LIN {X 0,Y 474.623,Z 516.173,A -85,B 0,C 180,E1 -7329.647,E2 -7329.647} C_VEL
LIN {X 0,Y 474.639,Z 516.177,A -85,B 0,C 180,E1 -7332.93,E2 -7332.93} C_VEL
LIN {X 0,Y 474.612,Z 516.174,A -85,B 0,C 180,E1 -7335.896,E2 -7335.896} C_VEL
LIN {X 0,Y 474.638,Z 516.178,A -85,B 0,C 180,E1 -7339.038,E2 -7339.038} C_VEL
LIN {X 0,Y 474.613,Z 516.174,A -85,B 0,C 180,E1 -7341.702,E2 -7341.702} C_VEL
LIN {X 0,Y 474.623,Z 516.175,A -85,B 0,C 180,E1 -7344.726,E2 -7344.726} C_VEL
LIN {X 0,Y 474.629,Z 516.17,A -85,B 0,C 180,E1 -7347.788,E2 -7347.788} C_VEL
LIN {X 0,Y 474.624,Z 516.176,A -85,B 0,C 180,E1 -7350.882,E2 -7350.882} C_VEL
LIN {X 0,Y 474.657,Z 516.166,A -85,B 0,C 180,E1 -7353.628,E2 -7353.628} C_VEL
LIN {X 0,Y 474.626,Z 516.176,A -85,B 0,C 180,E1 -7356.641,E2 -7356.641} C_VEL
LIN {X 0,Y 474.647,Z 516.168,A -85,B 0,C 180,E1 -7360.09,E2 -7360.09} C_VEL
LIN {X 0,Y 474.642,Z 516.174,A -85,B 0,C 180,E1 -7362.774,E2 -7362.774} C_VEL
LIN {X 0,Y 474.639,Z 516.173,A -85,B 0,C 180,E1 -7365.421,E2 -7365.421} C_VEL
LIN {X 0,Y 474.729,Z 516.161,A -85,B 0,C 180,E1 -7368.038,E2 -7368.038} C_VEL
LIN {X 0,Y 474.719,Z 516.164,A -85,B 0,C 180,E1 -7371.487,E2 -7371.487} C_VEL
LIN {X 0,Y 474.782,Z 516.155,A -85,B 0,C 180,E1 -7374.053,E2 -7374.053} C_VEL
LIN {X 0,Y 474.887,Z 516.143,A -85,B 0,C 180,E1 -7377.456,E2 -7377.456} C_VEL
LIN {X 0,Y 474.868,Z 516.149,A -85,B 0,C 180,E1 -7380.848,E2 -7380.848} C_VEL
LIN {X 0,Y 474.887,Z 516.145,A -85,B 0,C 180,E1 -7382.545,E2 -7382.545} C_VEL
LIN {X 0,Y 474.812,Z 516.337,A -85,B 0,C 180,E1 -7385.681,E2 -7385.681} C_VEL
LIN {X 0,Y 475.062,Z 517.484,A -85,B 0,C 180,E1 -7385.825,E2 -7385.825} C_VEL
LIN {X 0,Y 477.086,Z 523.784,A -85,B 0,C 180,E1 -7385.999,E2 -7385.999} C_VEL
LIN {X 0,Y 477.175,Z 549.292,A -85,B 0,C 180,E1 -7386.422,E2 -7386.422} C_VEL
LIN {X 0,Y 477.132,Z 562.414,A -85,B 0,C 180,E1 -7386.821,E2 -7386.821} C_VEL
LIN {X 0,Y 477,Z 574.255,A -85,B 0,C 180,E1 -7387.354,E2 -7387.354} C_VEL
LIN {X 0,Y 476.726,Z 585.813,A -85,B 0,C 180,E1 -7388.051,E2 -7388.051} C_VEL
LIN {X 0,Y 476.425,Z 597.212,A -85,B 0,C 180,E1 -7388.937,E2 -7388.937} C_VEL
LIN {X 0,Y 476.088,Z 605.867,A -85,B 0,C 180,E1 -7389.774,E2 -7389.774} C_VEL
LIN {X 0,Y 475.715,Z 614.993,A -85,B 0,C 180,E1 -7390.858,E2 -7390.858} C_VEL
LIN {X 0,Y 475.355,Z 623.876,A -85,B 0,C 180,E1 -7392.172,E2 -7392.172} C_VEL
LIN {X 0,Y 475.083,Z 630.832,A -85,B 0,C 180,E1 -7393.474,E2 -7393.474} C_VEL
LIN {X 0,Y 474.877,Z 635.577,A -85,B 0,C 180,E1 -7394.572,E2 -7394.572} C_VEL
LIN {X 0,Y 474.662,Z 639.7,A -85,B 0,C 180,E1 -7395.765,E2 -7395.765} C_VEL
LIN {X 0,Y 474.47,Z 643.459,A -85,B 0,C 180,E1 -7397.233,E2 -7397.233} C_VEL
LIN {X 0,Y 474.398,Z 645.704,A -85,B 0,C 180,E1 -7398.539,E2 -7398.539} C_VEL
LIN {X 0,Y 474.307,Z 647.024,A -85,B 0,C 180,E1 -7399.926,E2 -7399.926} C_VEL
LIN {X 0,Y 474.28,Z 647.331,A -85,B 0,C 180,E1 -7401.009,E2 -7401.009} C_VEL
LIN {X 0,Y 474.283,Z 647.161,A -85,B 0,C 180,E1 -7401.744,E2 -7401.744} C_VEL
LIN {X 0,Y 474.298,Z 645.84,A -85,B 0,C 180,E1 -7403.267,E2 -7403.267} C_VEL
LIN {X 0,Y 474.483,Z 642.883,A -85,B 0,C 180,E1 -7404.945,E2 -7404.945} C_VEL
LIN {X 0,Y 474.631,Z 639.027,A -85,B 0,C 180,E1 -7406.374,E2 -7406.374} C_VEL
LIN {X 0,Y 474.799,Z 633.826,A -85,B 0,C 180,E1 -7407.792,E2 -7407.792} C_VEL
LIN {X 0,Y 475.057,Z 627.036,A -85,B 0,C 180,E1 -7409.223,E2 -7409.223} C_VEL
LIN {X 0,Y 475.375,Z 619.877,A -85,B 0,C 180,E1 -7410.42,E2 -7410.42} C_VEL
LIN {X 0,Y 475.707,Z 610.882,A -85,B 0,C 180,E1 -7411.633,E2 -7411.633} C_VEL
LIN {X 0,Y 476.098,Z 600.971,A -85,B 0,C 180,E1 -7412.712,E2 -7412.712} C_VEL
LIN {X 0,Y 476.452,Z 591.039,A -85,B 0,C 180,E1 -7413.584,E2 -7413.584} C_VEL
LIN {X 0,Y 476.762,Z 579.896,A -85,B 0,C 180,E1 -7414.363,E2 -7414.363} C_VEL
LIN {X 0,Y 477.01,Z 567.71,A -85,B 0,C 180,E1 -7415.02,E2 -7415.02} C_VEL
LIN {X 0,Y 477.163,Z 555.29,A -85,B 0,C 180,E1 -7415.506,E2 -7415.506} C_VEL
LIN {X 0,Y 477.222,Z 541.716,A -85,B 0,C 180,E1 -7415.841,E2 -7415.841} C_VEL
LIN {X 0,Y 477.132,Z 524.228,A -85,B 0,C 180,E1 -7416.121,E2 -7416.121} C_VEL
LIN {X 0,Y 474.794,Z 517.041,A -85,B 0,C 180,E1 -7416.335,E2 -7416.335} C_VEL
LIN {X 0,Y 474.628,Z 516.233,A -85,B 0,C 180,E1 -7416.518,E2 -7416.518} C_VEL
LIN {X 0,Y 474.624,Z 516.178,A -85,B 0,C 180,E1 -7419.649,E2 -7419.649} C_VEL
LIN {X 0,Y 474.632,Z 516.175,A -85,B 0,C 180,E1 -7422.933,E2 -7422.933} C_VEL
LIN {X 0,Y 474.616,Z 516.174,A -85,B 0,C 180,E1 -7425.897,E2 -7425.897} C_VEL
LIN {X 0,Y 474.644,Z 516.172,A -85,B 0,C 180,E1 -7429.039,E2 -7429.039} C_VEL
LIN {X 0,Y 474.615,Z 516.177,A -85,B 0,C 180,E1 -7431.704,E2 -7431.704} C_VEL
LIN {X 0,Y 474.57,Z 516.182,A -85,B 0,C 180,E1 -7433.223,E2 -7433.223} C_VEL
LIN {X 0,Y 473.912,Z 516.264,A -85,B 0,C 180,E1 -7433.932,E2 -7433.932} C_VEL
LIN {X 0,Y 471.063,Z 516.618,A -85,B 0,C 180,E1 -7435.083,E2 -7435.083} C_VEL
LIN {X 0,Y 468.66,Z 516.916,A -85,B 0,C 180,E1 -7436.012,E2 -7436.012} C_VEL
LIN {X 0,Y 467.644,Z 517.042,A -85,B 0,C 180,E1 -7436.729,E2 -7436.729} C_VEL
LIN {X 0,Y 467.57,Z 517.052,A -85,B 0,C 180,E1 -7436.972,E2 -7436.972} C_VEL
LIN {X 0,Y 467.571,Z 517.055,A -85,B 0,C 180,E1 -7439.267,E2 -7439.267} C_VEL
LIN {X 0,Y 467.647,Z 517.04,A -85,B 0,C 180,E1 -7442.46,E2 -7442.46} C_VEL
LIN {X 0,Y 467.604,Z 517.049,A -85,B 0,C 180,E1 -7445.113,E2 -7445.113} C_VEL
LIN {X 0,Y 467.537,Z 517.057,A -85,B 0,C 180,E1 -7447.927,E2 -7447.927} C_VEL
LIN {X 0,Y 467.625,Z 517.043,A -85,B 0,C 180,E1 -7450.693,E2 -7450.693} C_VEL
LIN {X 0,Y 467.643,Z 517.042,A -85,B 0,C 180,E1 -7454.306,E2 -7454.306} C_VEL
LIN {X 0,Y 467.66,Z 517.044,A -85,B 0,C 180,E1 -7457.855,E2 -7457.855} C_VEL
LIN {X 0,Y 467.685,Z 517.04,A -85,B 0,C 180,E1 -7461.358,E2 -7461.358} C_VEL
LIN {X 0,Y 467.725,Z 517.035,A -85,B 0,C 180,E1 -7463.963,E2 -7463.963} C_VEL
LIN {X 0,Y 467.863,Z 517.018,A -85,B 0,C 180,E1 -7467.417,E2 -7467.417} C_VEL
LIN {X 0,Y 467.887,Z 517.015,A -85,B 0,C 180,E1 -7470,E2 -7470} C_VEL
LIN {X 0,Y 467.864,Z 517.013,A -85,B 0,C 180,E1 -7472.583,E2 -7472.583} C_VEL
LIN {X 0,Y 467.726,Z 517.036,A -85,B 0,C 180,E1 -7476.038,E2 -7476.038} C_VEL
LIN {X 0,Y 467.667,Z 517.042,A -85,B 0,C 180,E1 -7479.515,E2 -7479.515} C_VEL
LIN {X 0,Y 467.659,Z 517.041,A -85,B 0,C 180,E1 -7482.357,E2 -7482.357} C_VEL
LIN {X 0,Y 467.654,Z 517.048,A -85,B 0,C 180,E1 -7485.885,E2 -7485.885} C_VEL
LIN {X 0,Y 467.627,Z 517.044,A -85,B 0,C 180,E1 -7489.307,E2 -7489.307} C_VEL
LIN {X 0,Y 467.538,Z 517.06,A -85,B 0,C 180,E1 -7492.073,E2 -7492.073} C_VEL
LIN {X 0,Y 467.588,Z 517.048,A -85,B 0,C 180,E1 -7494.888,E2 -7494.888} C_VEL
LIN {X 0,Y 467.622,Z 517.049,A -85,B 0,C 180,E1 -7497.768,E2 -7497.768} C_VEL
LIN {X 0,Y 467.569,Z 517.05,A -85,B 0,C 180,E1 -7501.044,E2 -7501.044} C_VEL
LIN {X 0,Y 467.589,Z 517.053,A -85,B 0,C 180,E1 -7504.241,E2 -7504.241} C_VEL
LIN {X 0,Y 467.548,Z 517.053,A -85,B 0,C 180,E1 -7507.185,E2 -7507.185} C_VEL
LIN {X 0,Y 467.596,Z 517.053,A -85,B 0,C 180,E1 -7510.262,E2 -7510.262} C_VEL
LIN {X 0,Y 467.618,Z 517.046,A -85,B 0,C 180,E1 -7512.57,E2 -7512.57} C_VEL
LIN {X 0,Y 467.568,Z 517.05,A -85,B 0,C 180,E1 -7515.052,E2 -7515.052} C_VEL
LIN {X 0,Y 467.586,Z 517.049,A -85,B 0,C 180,E1 -7517.439,E2 -7517.439} C_VEL
LIN {X 0,Y 467.579,Z 517.05,A -85,B 0,C 180,E1 -7520.854,E2 -7520.854} C_VEL
LIN {X 0,Y 467.559,Z 517.059,A -85,B 0,C 180,E1 -7524.259,E2 -7524.259} C_VEL
LIN {X 0,Y 467.578,Z 517.049,A -85,B 0,C 180,E1 -7527.32,E2 -7527.32} C_VEL
LIN {X 0,Y 467.573,Z 517.052,A -85,B 0,C 180,E1 -7530.665,E2 -7530.665} C_VEL
LIN {X 0,Y 467.621,Z 517.043,A -85,B 0,C 180,E1 -7533.2,E2 -7533.2} C_VEL
LIN {X 0,Y 467.586,Z 517.054,A -85,B 0,C 180,E1 -7536.467,E2 -7536.467} C_VEL
LIN {X 0,Y 467.617,Z 517.046,A -85,B 0,C 180,E1 -7539.777,E2 -7539.777} C_VEL
LIN {X 0,Y 467.602,Z 517.052,A -85,B 0,C 180,E1 -7542.506,E2 -7542.506} C_VEL
LIN {X 0,Y 467.598,Z 517.047,A -85,B 0,C 180,E1 -7545.196,E2 -7545.196} C_VEL
LIN {X 0,Y 467.674,Z 517.039,A -85,B 0,C 180,E1 -7547.855,E2 -7547.855} C_VEL
LIN {X 0,Y 467.674,Z 517.037,A -85,B 0,C 180,E1 -7551.357,E2 -7551.357} C_VEL
LIN {X 0,Y 467.743,Z 517.031,A -85,B 0,C 180,E1 -7553.962,E2 -7553.962} C_VEL
LIN {X 0,Y 467.852,Z 517.015,A -85,B 0,C 180,E1 -7557.417,E2 -7557.417} C_VEL
LIN {X 0,Y 467.873,Z 517.014,A -85,B 0,C 180,E1 -7560,E2 -7560} C_VEL
LIN {X 0,Y 467.852,Z 517.022,A -85,B 0,C 180,E1 -7562.583,E2 -7562.583} C_VEL
LIN {X 0,Y 467.735,Z 517.032,A -85,B 0,C 180,E1 -7566.037,E2 -7566.037} C_VEL
LIN {X 0,Y 467.673,Z 517.044,A -85,B 0,C 180,E1 -7568.643,E2 -7568.643} C_VEL
LIN {X 0,Y 467.646,Z 517.043,A -85,B 0,C 180,E1 -7572.145,E2 -7572.145} C_VEL
LIN {X 0,Y 467.63,Z 517.042,A -85,B 0,C 180,E1 -7575.695,E2 -7575.695} C_VEL
LIN {X 0,Y 467.609,Z 517.052,A -85,B 0,C 180,E1 -7578.765,E2 -7578.765} C_VEL
LIN {X 0,Y 467.572,Z 517.051,A -85,B 0,C 180,E1 -7581.269,E2 -7581.269} C_VEL
LIN {X 0,Y 467.564,Z 517.051,A -85,B 0,C 180,E1 -7583.943,E2 -7583.943} C_VEL
LIN {X 0,Y 467.62,Z 517.051,A -85,B 0,C 180,E1 -7586.8,E2 -7586.8} C_VEL
LIN {X 0,Y 467.579,Z 517.049,A -85,B 0,C 180,E1 -7589.736,E2 -7589.736} C_VEL
LIN {X 0,Y 467.576,Z 517.058,A -85,B 0,C 180,E1 -7592.759,E2 -7592.759} C_VEL
LIN {X 0,Y 467.55,Z 517.052,A -85,B 0,C 180,E1 -7595.89,E2 -7595.89} C_VEL
LIN {X 0,Y 467.576,Z 517.053,A -85,B 0,C 180,E1 -7599.145,E2 -7599.145} C_VEL
LIN {X 0,Y 467.58,Z 517.053,A -85,B 0,C 180,E1 -7602.567,E2 -7602.567} C_VEL
LIN {X 0,Y 467.565,Z 517.056,A -85,B 0,C 180,E1 -7605.054,E2 -7605.054} C_VEL
LIN {X 0,Y 467.584,Z 517.05,A -85,B 0,C 180,E1 -7607.44,E2 -7607.44} C_VEL
LIN {X 0,Y 467.58,Z 517.057,A -85,B 0,C 180,E1 -7610.856,E2 -7610.856} C_VEL
LIN {X 0,Y 467.558,Z 517.054,A -85,B 0,C 180,E1 -7614.261,E2 -7614.261} C_VEL
LIN {X 0,Y 467.579,Z 517.057,A -85,B 0,C 180,E1 -7617.321,E2 -7617.321} C_VEL
LIN {X 0,Y 467.62,Z 517.228,A -85,B 0,C 180,E1 -7618.944,E2 -7618.944} C_VEL
LIN {X 0,Y 470.423,Z 531.107,A -85,B 0,C 180,E1 -7621.678,E2 -7621.678} C_VEL
LIN {X 0,Y 470.116,Z 540.418,A -85,B 0,C 180,E1 -7623.354,E2 -7623.354} C_VEL
LIN {X 0,Y 469.299,Z 558.979,A -85,B 0,C 180,E1 -7626.619,E2 -7626.619} C_VEL
LIN {X 0,Y 468.488,Z 577.522,A -85,B 0,C 180,E1 -7629.817,E2 -7629.817} C_VEL
LIN {X 0,Y 468.046,Z 592.113,A -85,B 0,C 180,E1 -7632.298,E2 -7632.298} C_VEL
LIN {X 0,Y 467.637,Z 610.659,A -85,B 0,C 180,E1 -7635.42,E2 -7635.42} C_VEL
LIN {X 0,Y 467.447,Z 616.633,A -85,B 0,C 180,E1 -7636.386,E2 -7636.386} C_VEL
LIN {X 0,Y 469.563,Z 640.275,A -85,B 0,C 180,E1 -7636.878,E2 -7636.878} C_VEL
LIN {X 0,Y 469.124,Z 698.067,A -85,B 0,C 180,E1 -7637.871,E2 -7637.871} C_VEL
LIN {X 0,Y 468.748,Z 709.114,A -85,B 0,C 180,E1 -7638.213,E2 -7638.213} C_VEL
LIN {X 0,Y 468.397,Z 720.606,A -85,B 0,C 180,E1 -7638.752,E2 -7638.752} C_VEL
LIN {X 0,Y 468.018,Z 730.817,A -85,B 0,C 180,E1 -7639.4,E2 -7639.4} C_VEL
LIN {X 0,Y 467.616,Z 741.243,A -85,B 0,C 180,E1 -7640.266,E2 -7640.266} C_VEL
LIN {X 0,Y 467.318,Z 749.497,A -85,B 0,C 180,E1 -7641.133,E2 -7641.133} C_VEL
LIN {X 0,Y 467.121,Z 757.771,A -85,B 0,C 180,E1 -7642.218,E2 -7642.218} C_VEL
LIN {X 0,Y 467.063,Z 764.185,A -85,B 0,C 180,E1 -7643.272,E2 -7643.272} C_VEL
LIN {X 0,Y 466.964,Z 769.568,A -85,B 0,C 180,E1 -7644.386,E2 -7644.386} C_VEL
LIN {X 0,Y 466.953,Z 774.391,A -85,B 0,C 180,E1 -7645.684,E2 -7645.684} C_VEL
LIN {X 0,Y 466.975,Z 776.783,A -85,B 0,C 180,E1 -7646.549,E2 -7646.549} C_VEL
LIN {X 0,Y 466.93,Z 778.604,A -85,B 0,C 180,E1 -7647.412,E2 -7647.412} C_VEL
LIN {X 0,Y 466.913,Z 779.879,A -85,B 0,C 180,E1 -7648.275,E2 -7648.275} C_VEL
LIN {X 0,Y 466.917,Z 780.608,A -85,B 0,C 180,E1 -7649.138,E2 -7649.138} C_VEL
LIN {X 0,Y 467.053,Z 780.859,A -85,B 0,C 180,E1 -7650,E2 -7650} C_VEL
LIN {X 0,Y 466.929,Z 780.514,A -85,B 0,C 180,E1 -7650.862,E2 -7650.862} C_VEL
LIN {X 0,Y 466.936,Z 779.7,A -85,B 0,C 180,E1 -7651.725,E2 -7651.725} C_VEL
LIN {X 0,Y 466.961,Z 778.321,A -85,B 0,C 180,E1 -7652.588,E2 -7652.588} C_VEL
LIN {X 0,Y 467.012,Z 775.24,A -85,B 0,C 180,E1 -7653.883,E2 -7653.883} C_VEL
LIN {X 0,Y 466.958,Z 770.741,A -85,B 0,C 180,E1 -7655.181,E2 -7655.181} C_VEL
LIN {X 0,Y 467.062,Z 764.905,A -85,B 0,C 180,E1 -7656.445,E2 -7656.445} C_VEL
LIN {X 0,Y 467.113,Z 758.249,A -85,B 0,C 180,E1 -7657.565,E2 -7657.565} C_VEL
LIN {X 0,Y 467.283,Z 750.162,A -85,B 0,C 180,E1 -7658.65,E2 -7658.65} C_VEL
LIN {X 0,Y 467.545,Z 740.997,A -85,B 0,C 180,E1 -7659.626,E2 -7659.626} C_VEL
LIN {X 0,Y 467.91,Z 730.624,A -85,B 0,C 180,E1 -7660.493,E2 -7660.493} C_VEL
LIN {X 0,Y 468.299,Z 719.691,A -85,B 0,C 180,E1 -7661.195,E2 -7661.195} C_VEL
LIN {X 0,Y 468.652,Z 708.238,A -85,B 0,C 180,E1 -7661.735,E2 -7661.735} C_VEL
LIN {X 0,Y 469.06,Z 696.256,A -85,B 0,C 180,E1 -7662.108,E2 -7662.108} C_VEL
LIN {X 0,Y 469.386,Z 644.85,A -85,B 0,C 180,E1 -7662.978,E2 -7662.978} C_VEL
LIN {X 0,Y 469.097,Z 635.875,A -85,B 0,C 180,E1 -7663.138,E2 -7663.138} C_VEL
LIN {X 0,Y 467.424,Z 613.413,A -85,B 0,C 180,E1 -7663.587,E2 -7663.587} C_VEL
LIN {X 0,Y 467.456,Z 610.902,A -85,B 0,C 180,E1 -7663.919,E2 -7663.919} C_VEL
LIN {X 0,Y 467.813,Z 590.403,A -85,B 0,C 180,E1 -7667.259,E2 -7667.259} C_VEL
LIN {X 0,Y 468.259,Z 569.924,A -85,B 0,C 180,E1 -7670.652,E2 -7670.652} C_VEL
LIN {X 0,Y 468.806,Z 550.911,A -85,B 0,C 180,E1 -7673.876,E2 -7673.876} C_VEL
LIN {X 0,Y 469.473,Z 532.108,A -85,B 0,C 180,E1 -7677.166,E2 -7677.166} C_VEL
LIN {X 0,Y 469.564,Z 527.557,A -85,B 0,C 180,E1 -7677.987,E2 -7677.987} C_VEL
LIN {X 0,Y 467.63,Z 517.169,A -85,B 0,C 180,E1 -7680.042,E2 -7680.042} C_VEL
LIN {X 0,Y 467.58,Z 517.056,A -85,B 0,C 180,E1 -7682.758,E2 -7682.758} C_VEL
LIN {X 0,Y 467.551,Z 517.055,A -85,B 0,C 180,E1 -7685.889,E2 -7685.889} C_VEL
LIN {X 0,Y 467.578,Z 517.056,A -85,B 0,C 180,E1 -7689.144,E2 -7689.144} C_VEL
LIN {X 0,Y 467.58,Z 517.052,A -85,B 0,C 180,E1 -7692.566,E2 -7692.566} C_VEL
LIN {X 0,Y 467.564,Z 517.056,A -85,B 0,C 180,E1 -7695.053,E2 -7695.053} C_VEL
LIN {X 0,Y 467.618,Z 517.044,A -85,B 0,C 180,E1 -7697.443,E2 -7697.443} C_VEL
LIN {X 0,Y 467.612,Z 517.049,A -85,B 0,C 180,E1 -7700.858,E2 -7700.858} C_VEL
LIN {X 0,Y 467.556,Z 517.052,A -85,B 0,C 180,E1 -7704.26,E2 -7704.26} C_VEL
LIN {X 0,Y 467.574,Z 517.052,A -85,B 0,C 180,E1 -7707.32,E2 -7707.32} C_VEL
LIN {X 0,Y 467.57,Z 517.054,A -85,B 0,C 180,E1 -7710.665,E2 -7710.665} C_VEL
LIN {X 0,Y 467.619,Z 517.046,A -85,B 0,C 180,E1 -7713.2,E2 -7713.2} C_VEL
LIN {X 0,Y 467.583,Z 517.052,A -85,B 0,C 180,E1 -7716.468,E2 -7716.468} C_VEL
LIN {X 0,Y 467.614,Z 517.044,A -85,B 0,C 180,E1 -7719.777,E2 -7719.777} C_VEL
LIN {X 0,Y 467.6,Z 517.05,A -85,B 0,C 180,E1 -7722.507,E2 -7722.507} C_VEL
LIN {X 0,Y 467.597,Z 517.053,A -85,B 0,C 180,E1 -7725.196,E2 -7725.196} C_VEL
LIN {X 0,Y 467.687,Z 517.038,A -85,B 0,C 180,E1 -7727.856,E2 -7727.856} C_VEL
LIN {X 0,Y 467.673,Z 517.043,A -85,B 0,C 180,E1 -7731.357,E2 -7731.357} C_VEL
LIN {X 0,Y 467.744,Z 517.032,A -85,B 0,C 180,E1 -7733.963,E2 -7733.963} C_VEL
LIN {X 0,Y 467.852,Z 517.02,A -85,B 0,C 180,E1 -7737.417,E2 -7737.417} C_VEL
LIN {X 0,Y 467.873,Z 517.016,A -85,B 0,C 180,E1 -7740,E2 -7740} C_VEL
LIN {X 0,Y 467.852,Z 517.021,A -85,B 0,C 180,E1 -7742.583,E2 -7742.583} C_VEL
LIN {X 0,Y 467.76,Z 517.165,A -85,B 0,C 180,E1 -7745.443,E2 -7745.443} C_VEL
LIN {X 0,Y 467.998,Z 518.237,A -85,B 0,C 180,E1 -7745.602,E2 -7745.602} C_VEL
LIN {X 0,Y 470.331,Z 525.484,A -85,B 0,C 180,E1 -7745.803,E2 -7745.803} C_VEL
LIN {X 0,Y 470.316,Z 550.256,A -85,B 0,C 180,E1 -7746.22,E2 -7746.22} C_VEL
LIN {X 0,Y 470.277,Z 563.453,A -85,B 0,C 180,E1 -7746.624,E2 -7746.624} C_VEL
LIN {X 0,Y 470.145,Z 575.827,A -85,B 0,C 180,E1 -7747.192,E2 -7747.192} C_VEL
LIN {X 0,Y 469.824,Z 588.1,A -85,B 0,C 180,E1 -7747.954,E2 -7747.954} C_VEL
LIN {X 0,Y 469.566,Z 598.1,A -85,B 0,C 180,E1 -7748.752,E2 -7748.752} C_VEL
LIN {X 0,Y 469.156,Z 607.733,A -85,B 0,C 180,E1 -7749.702,E2 -7749.702} C_VEL
LIN {X 0,Y 468.807,Z 616.704,A -85,B 0,C 180,E1 -7750.801,E2 -7750.801} C_VEL
LIN {X 0,Y 468.4,Z 625.436,A -85,B 0,C 180,E1 -7752.126,E2 -7752.126} C_VEL
LIN {X 0,Y 468.104,Z 632.319,A -85,B 0,C 180,E1 -7753.457,E2 -7753.457} C_VEL
LIN {X 0,Y 467.852,Z 637.784,A -85,B 0,C 180,E1 -7754.796,E2 -7754.796} C_VEL
LIN {X 0,Y 467.635,Z 641.308,A -85,B 0,C 180,E1 -7755.883,E2 -7755.883} C_VEL
LIN {X 0,Y 467.454,Z 645.129,A -85,B 0,C 180,E1 -7757.5,E2 -7757.5} C_VEL
LIN {X 0,Y 467.376,Z 646.948,A -85,B 0,C 180,E1 -7758.681,E2 -7758.681} C_VEL
LIN {X 0,Y 467.289,Z 648.199,A -85,B 0,C 180,E1 -7760.238,E2 -7760.238} C_VEL
LIN {X 0,Y 467.263,Z 648.317,A -85,B 0,C 180,E1 -7761.171,E2 -7761.171} C_VEL
LIN {X 0,Y 467.254,Z 647.963,A -85,B 0,C 180,E1 -7762.088,E2 -7762.088} C_VEL
LIN {X 0,Y 467.285,Z 646.625,A -85,B 0,C 180,E1 -7763.448,E2 -7763.448} C_VEL
LIN {X 0,Y 467.451,Z 644.073,A -85,B 0,C 180,E1 -7764.896,E2 -7764.896} C_VEL
LIN {X 0,Y 467.619,Z 640.383,A -85,B 0,C 180,E1 -7766.319,E2 -7766.319} C_VEL
LIN {X 0,Y 467.806,Z 635.294,A -85,B 0,C 180,E1 -7767.757,E2 -7767.757} C_VEL
LIN {X 0,Y 468.037,Z 629.218,A -85,B 0,C 180,E1 -7769.09,E2 -7769.09} C_VEL
LIN {X 0,Y 468.386,Z 621.573,A -85,B 0,C 180,E1 -7770.425,E2 -7770.425} C_VEL
LIN {X 0,Y 468.74,Z 612.773,A -85,B 0,C 180,E1 -7771.653,E2 -7771.653} C_VEL
LIN {X 0,Y 469.139,Z 602.841,A -85,B 0,C 180,E1 -7772.767,E2 -7772.767} C_VEL
LIN {X 0,Y 469.496,Z 593.334,A -85,B 0,C 180,E1 -7773.633,E2 -7773.633} C_VEL
LIN {X 0,Y 469.831,Z 581.764,A -85,B 0,C 180,E1 -7774.475,E2 -7774.475} C_VEL
LIN {X 0,Y 470.109,Z 569.848,A -85,B 0,C 180,E1 -7775.139,E2 -7775.139} C_VEL
LIN {X 0,Y 470.277,Z 556.846,A -85,B 0,C 180,E1 -7775.669,E2 -7775.669} C_VEL
LIN {X 0,Y 470.314,Z 543.458,A -85,B 0,C 180,E1 -7776.013,E2 -7776.013} C_VEL
LIN {X 0,Y 470.23,Z 525.469,A -85,B 0,C 180,E1 -7776.312,E2 -7776.312} C_VEL
LIN {X 0,Y 467.743,Z 517.998,A -85,B 0,C 180,E1 -7776.528,E2 -7776.528} C_VEL
LIN {X 0,Y 467.563,Z 517.133,A -85,B 0,C 180,E1 -7776.701,E2 -7776.701} C_VEL
LIN {X 0,Y 467.579,Z 517.054,A -85,B 0,C 180,E1 -7779.956,E2 -7779.956} C_VEL
LIN {X 0,Y 467.583,Z 517.051,A -85,B 0,C 180,E1 -7782.568,E2 -7782.568} C_VEL
LIN {X 0,Y 467.568,Z 517.054,A -85,B 0,C 180,E1 -7785.054,E2 -7785.054} C_VEL
LIN {X 0,Y 467.622,Z 517.051,A -85,B 0,C 180,E1 -7787.445,E2 -7787.445} C_VEL
LIN {X 0,Y 467.614,Z 517.046,A -85,B 0,C 180,E1 -7790.86,E2 -7790.86} C_VEL
LIN {X 0,Y 467.559,Z 517.052,A -85,B 0,C 180,E1 -7794.262,E2 -7794.262} C_VEL
LIN {X 0,Y 467.57,Z 517.052,A -85,B 0,C 180,E1 -7796.972,E2 -7796.972} C_VEL
LIN {X 0,Y 466.932,Z 517.138,A -85,B 0,C 180,E1 -7797.69,E2 -7797.69} C_VEL
LIN {X 0,Y 464.104,Z 517.49,A -85,B 0,C 180,E1 -7798.857,E2 -7798.857} C_VEL
LIN {X 0,Y 461.688,Z 517.788,A -85,B 0,C 180,E1 -7799.798,E2 -7799.798} C_VEL
LIN {X 0,Y 460.634,Z 517.916,A -85,B 0,C 180,E1 -7800.525,E2 -7800.525} C_VEL
LIN {X 0,Y 460.541,Z 517.926,A -85,B 0,C 180,E1 -7800.771,E2 -7800.771} C_VEL
LIN {X 0,Y 460.565,Z 517.928,A -85,B 0,C 180,E1 -7803.736,E2 -7803.736} C_VEL
LIN {X 0,Y 460.548,Z 517.925,A -85,B 0,C 180,E1 -7806.625,E2 -7806.625} C_VEL
LIN {X 0,Y 460.554,Z 517.931,A -85,B 0,C 180,E1 -7809.453,E2 -7809.453} C_VEL
LIN {X 0,Y 460.553,Z 517.925,A -85,B 0,C 180,E1 -7812.23,E2 -7812.23} C_VEL
LIN {X 0,Y 460.569,Z 517.923,A -85,B 0,C 180,E1 -7814.965,E2 -7814.965} C_VEL
LIN {X 0,Y 460.615,Z 517.916,A -85,B 0,C 180,E1 -7818.56,E2 -7818.56} C_VEL
LIN {X 0,Y 460.671,Z 517.912,A -85,B 0,C 180,E1 -7822.108,E2 -7822.108} C_VEL
LIN {X 0,Y 460.693,Z 517.906,A -85,B 0,C 180,E1 -7824.748,E2 -7824.748} C_VEL
LIN {X 0,Y 460.804,Z 517.897,A -85,B 0,C 180,E1 -7827.378,E2 -7827.378} C_VEL
LIN {X 0,Y 460.858,Z 517.891,A -85,B 0,C 180,E1 -7830,E2 -7830} C_VEL
LIN {X 0,Y 460.805,Z 517.893,A -85,B 0,C 180,E1 -7832.622,E2 -7832.622} C_VEL
LIN {X 0,Y 460.69,Z 517.911,A -85,B 0,C 180,E1 -7836.13,E2 -7836.13} C_VEL
LIN {X 0,Y 460.625,Z 517.915,A -85,B 0,C 180,E1 -7838.776,E2 -7838.776} C_VEL
LIN {X 0,Y 460.618,Z 517.917,A -85,B 0,C 180,E1 -7842.445,E2 -7842.445} C_VEL
LIN {X 0,Y 460.604,Z 517.924,A -85,B 0,C 180,E1 -7845.997,E2 -7845.997} C_VEL
LIN {X 0,Y 460.575,Z 517.921,A -85,B 0,C 180,E1 -7848.901,E2 -7848.901} C_VEL
LIN {X 0,Y 460.519,Z 517.931,A -85,B 0,C 180,E1 -7851.485,E2 -7851.485} C_VEL
LIN {X 0,Y 460.534,Z 517.93,A -85,B 0,C 180,E1 -7854.332,E2 -7854.332} C_VEL
LIN {X 0,Y 460.573,Z 517.922,A -85,B 0,C 180,E1 -7857.243,E2 -7857.243} C_VEL
LIN {X 0,Y 460.512,Z 517.934,A -85,B 0,C 180,E1 -7860.239,E2 -7860.239} C_VEL
LIN {X 0,Y 460.53,Z 517.928,A -85,B 0,C 180,E1 -7863.324,E2 -7863.324} C_VEL
LIN {X 0,Y 460.476,Z 517.936,A -85,B 0,C 180,E1 -7866.529,E2 -7866.529} C_VEL
LIN {X 0,Y 460.574,Z 517.927,A -85,B 0,C 180,E1 -7869.857,E2 -7869.857} C_VEL
LIN {X 0,Y 460.541,Z 517.926,A -85,B 0,C 180,E1 -7872.903,E2 -7872.903} C_VEL
LIN {X 0,Y 460.509,Z 517.934,A -85,B 0,C 180,E1 -7875.829,E2 -7875.829} C_VEL
LIN {X 0,Y 460.528,Z 517.927,A -85,B 0,C 180,E1 -7878.988,E2 -7878.988} C_VEL
LIN {X 0,Y 460.523,Z 517.928,A -85,B 0,C 180,E1 -7881.266,E2 -7881.266} C_VEL
LIN {X 0,Y 460.509,Z 517.933,A -85,B 0,C 180,E1 -7884.554,E2 -7884.554} C_VEL
LIN {X 0,Y 460.528,Z 517.929,A -85,B 0,C 180,E1 -7887.715,E2 -7887.715} C_VEL
LIN {X 0,Y 460.542,Z 517.927,A -85,B 0,C 180,E1 -7890.769,E2 -7890.769} C_VEL
LIN {X 0,Y 460.562,Z 517.925,A -85,B 0,C 180,E1 -7893.734,E2 -7893.734} C_VEL
LIN {X 0,Y 460.539,Z 517.93,A -85,B 0,C 180,E1 -7896.623,E2 -7896.623} C_VEL
LIN {X 0,Y 460.545,Z 517.925,A -85,B 0,C 180,E1 -7899.452,E2 -7899.452} C_VEL
LIN {X 0,Y 460.552,Z 517.931,A -85,B 0,C 180,E1 -7902.23,E2 -7902.23} C_VEL
LIN {X 0,Y 460.557,Z 517.925,A -85,B 0,C 180,E1 -7904.964,E2 -7904.964} C_VEL
LIN {X 0,Y 460.621,Z 517.916,A -85,B 0,C 180,E1 -7907.666,E2 -7907.666} C_VEL
LIN {X 0,Y 460.621,Z 517.916,A -85,B 0,C 180,E1 -7911.223,E2 -7911.223} C_VEL
LIN {X 0,Y 460.708,Z 517.906,A -85,B 0,C 180,E1 -7913.87,E2 -7913.87} C_VEL
LIN {X 0,Y 460.817,Z 517.891,A -85,B 0,C 180,E1 -7917.377,E2 -7917.377} C_VEL
LIN {X 0,Y 460.844,Z 517.89,A -85,B 0,C 180,E1 -7920,E2 -7920} C_VEL
LIN {X 0,Y 460.817,Z 517.898,A -85,B 0,C 180,E1 -7922.622,E2 -7922.622} C_VEL
LIN {X 0,Y 460.701,Z 517.909,A -85,B 0,C 180,E1 -7926.13,E2 -7926.13} C_VEL
LIN {X 0,Y 460.62,Z 517.921,A -85,B 0,C 180,E1 -7928.776,E2 -7928.776} C_VEL
LIN {X 0,Y 460.604,Z 517.924,A -85,B 0,C 180,E1 -7932.445,E2 -7932.445} C_VEL
LIN {X 0,Y 460.591,Z 517.92,A -85,B 0,C 180,E1 -7935.998,E2 -7935.998} C_VEL
LIN {X 0,Y 460.562,Z 517.928,A -85,B 0,C 180,E1 -7938.902,E2 -7938.902} C_VEL
LIN {X 0,Y 460.507,Z 517.93,A -85,B 0,C 180,E1 -7941.486,E2 -7941.486} C_VEL
LIN {X 0,Y 460.534,Z 517.93,A -85,B 0,C 180,E1 -7944.332,E2 -7944.332} C_VEL
LIN {X 0,Y 460.576,Z 517.923,A -85,B 0,C 180,E1 -7947.243,E2 -7947.243} C_VEL
LIN {X 0,Y 460.52,Z 517.93,A -85,B 0,C 180,E1 -7950.239,E2 -7950.239} C_VEL
LIN {X 0,Y 460.522,Z 517.93,A -85,B 0,C 180,E1 -7953.325,E2 -7953.325} C_VEL
LIN {X 0,Y 460.472,Z 517.939,A -85,B 0,C 180,E1 -7956.53,E2 -7956.53} C_VEL
LIN {X 0,Y 460.538,Z 517.933,A -85,B 0,C 180,E1 -7958.898,E2 -7958.898} C_VEL
LIN {X 0,Y 460.518,Z 517.929,A -85,B 0,C 180,E1 -7962.182,E2 -7962.182} C_VEL
LIN {X 0,Y 460.515,Z 517.93,A -85,B 0,C 180,E1 -7965.412,E2 -7965.412} C_VEL
LIN {X 0,Y 460.53,Z 517.929,A -85,B 0,C 180,E1 -7968.398,E2 -7968.398} C_VEL
LIN {X 0,Y 460.527,Z 517.931,A -85,B 0,C 180,E1 -7971.268,E2 -7971.268} C_VEL
LIN {X 0,Y 460.509,Z 517.935,A -85,B 0,C 180,E1 -7974.555,E2 -7974.555} C_VEL
LIN {X 0,Y 460.532,Z 517.933,A -85,B 0,C 180,E1 -7977.716,E2 -7977.716} C_VEL
LIN {X 0,Y 460.579,Z 518.159,A -85,B 0,C 180,E1 -7978.748,E2 -7978.748} C_VEL
LIN {X 0,Y 463.448,Z 532.352,A -85,B 0,C 180,E1 -7981.587,E2 -7981.587} C_VEL
LIN {X 0,Y 463.28,Z 539.644,A -85,B 0,C 180,E1 -7982.929,E2 -7982.929} C_VEL
LIN {X 0,Y 462.298,Z 559.467,A -85,B 0,C 180,E1 -7986.481,E2 -7986.481} C_VEL
LIN {X 0,Y 461.458,Z 577.955,A -85,B 0,C 180,E1 -7989.728,E2 -7989.728} C_VEL
LIN {X 0,Y 460.904,Z 595.124,A -85,B 0,C 180,E1 -7992.702,E2 -7992.702} C_VEL
LIN {X 0,Y 460.409,Z 613.57,A -85,B 0,C 180,E1 -7995.864,E2 -7995.864} C_VEL
LIN {X 0,Y 460.41,Z 615.765,A -85,B 0,C 180,E1 -7996.173,E2 -7996.173} C_VEL
LIN {X 0,Y 462.655,Z 641.477,A -85,B 0,C 180,E1 -7996.704,E2 -7996.704} C_VEL
LIN {X 0,Y 462.148,Z 697.14,A -85,B 0,C 180,E1 -7997.685,E2 -7997.685} C_VEL
LIN {X 0,Y 461.79,Z 708.124,A -85,B 0,C 180,E1 -7998.033,E2 -7998.033} C_VEL
LIN {X 0,Y 461.414,Z 719.591,A -85,B 0,C 180,E1 -7998.58,E2 -7998.58} C_VEL
LIN {X 0,Y 461.027,Z 729.799,A -85,B 0,C 180,E1 -7999.238,E2 -7999.238} C_VEL
LIN {X 0,Y 460.621,Z 740.227,A -85,B 0,C 180,E1 -8000.116,E2 -8000.116} C_VEL
LIN {X 0,Y 460.246,Z 748.478,A -85,B 0,C 180,E1 -8000.995,E2 -8000.995} C_VEL
LIN {X 0,Y 460.06,Z 756.761,A -85,B 0,C 180,E1 -8002.098,E2 -8002.098} C_VEL
LIN {X 0,Y 459.975,Z 763.785,A -85,B 0,C 180,E1 -8003.285,E2 -8003.285} C_VEL
LIN {X 0,Y 459.91,Z 768.573,A -85,B 0,C 180,E1 -8004.3,E2 -8004.3} C_VEL
LIN {X 0,Y 459.896,Z 773.402,A -85,B 0,C 180,E1 -8005.618,E2 -8005.618} C_VEL
LIN {X 0,Y 459.934,Z 775.798,A -85,B 0,C 180,E1 -8006.496,E2 -8006.496} C_VEL
LIN {X 0,Y 459.884,Z 777.62,A -85,B 0,C 180,E1 -8007.372,E2 -8007.372} C_VEL
LIN {X 0,Y 459.874,Z 778.894,A -85,B 0,C 180,E1 -8008.248,E2 -8008.248} C_VEL
LIN {X 0,Y 459.882,Z 779.623,A -85,B 0,C 180,E1 -8009.124,E2 -8009.124} C_VEL
LIN {X 0,Y 460.034,Z 779.87,A -85,B 0,C 180,E1 -8010,E2 -8010} C_VEL
LIN {X 0,Y 459.896,Z 779.518,A -85,B 0,C 180,E1 -8010.876,E2 -8010.876} C_VEL
LIN {X 0,Y 459.899,Z 778.694,A -85,B 0,C 180,E1 -8011.751,E2 -8011.751} C_VEL
LIN {X 0,Y 459.917,Z 777.304,A -85,B 0,C 180,E1 -8012.627,E2 -8012.627} C_VEL
LIN {X 0,Y 459.965,Z 774.207,A -85,B 0,C 180,E1 -8013.942,E2 -8013.942} C_VEL
LIN {X 0,Y 459.897,Z 769.681,A -85,B 0,C 180,E1 -8015.261,E2 -8015.261} C_VEL
LIN {X 0,Y 459.997,Z 764.302,A -85,B 0,C 180,E1 -8016.455,E2 -8016.455} C_VEL
LIN {X 0,Y 460.04,Z 757.155,A -85,B 0,C 180,E1 -8017.682,E2 -8017.682} C_VEL
LIN {X 0,Y 460.219,Z 749.058,A -85,B 0,C 180,E1 -8018.784,E2 -8018.784} C_VEL
LIN {X 0,Y 460.54,Z 739.894,A -85,B 0,C 180,E1 -8019.774,E2 -8019.774} C_VEL
LIN {X 0,Y 460.818,Z 730.991,A -85,B 0,C 180,E1 -8020.545,E2 -8020.545} C_VEL
LIN {X 0,Y 461.271,Z 719.589,A -85,B 0,C 180,E1 -8021.312,E2 -8021.312} C_VEL
LIN {X 0,Y 461.653,Z 708.516,A -85,B 0,C 180,E1 -8021.859,E2 -8021.859} C_VEL
LIN {X 0,Y 462.085,Z 696.567,A -85,B 0,C 180,E1 -8022.266,E2 -8022.266} C_VEL
LIN {X 0,Y 462.291,Z 678.528,A -85,B 0,C 180,E1 -8022.608,E2 -8022.608} C_VEL
LIN {X 0,Y 462.375,Z 638.236,A -85,B 0,C 180,E1 -8023.293,E2 -8023.293} C_VEL
LIN {X 0,Y 460.365,Z 611.855,A -85,B 0,C 180,E1 -8023.827,E2 -8023.827} C_VEL
LIN {X 0,Y 460.38,Z 609.529,A -85,B 0,C 180,E1 -8024.137,E2 -8024.137} C_VEL
LIN {X 0,Y 460.734,Z 590.468,A -85,B 0,C 180,E1 -8027.304,E2 -8027.304} C_VEL
LIN {X 0,Y 461.19,Z 570.074,A -85,B 0,C 180,E1 -8030.75,E2 -8030.75} C_VEL
LIN {X 0,Y 461.789,Z 550.97,A -85,B 0,C 180,E1 -8034.057,E2 -8034.057} C_VEL
LIN {X 0,Y 462.523,Z 532.482,A -85,B 0,C 180,E1 -8037.363,E2 -8037.363} C_VEL
LIN {X 0,Y 462.461,Z 528.057,A -85,B 0,C 180,E1 -8038.186,E2 -8038.186} C_VEL
LIN {X 0,Y 460.611,Z 518.233,A -85,B 0,C 180,E1 -8040.152,E2 -8040.152} C_VEL
LIN {X 0,Y 460.553,Z 517.931,A -85,B 0,C 180,E1 -8040.489,E2 -8040.489} C_VEL
LIN {X 0,Y 460.525,Z 517.934,A -85,B 0,C 180,E1 -8043.324,E2 -8043.324} C_VEL
LIN {X 0,Y 460.474,Z 517.94,A -85,B 0,C 180,E1 -8046.529,E2 -8046.529} C_VEL
LIN {X 0,Y 460.54,Z 517.933,A -85,B 0,C 180,E1 -8048.897,E2 -8048.897} C_VEL
LIN {X 0,Y 460.518,Z 517.93,A -85,B 0,C 180,E1 -8052.181,E2 -8052.181} C_VEL
LIN {X 0,Y 460.516,Z 517.933,A -85,B 0,C 180,E1 -8055.412,E2 -8055.412} C_VEL
LIN {X 0,Y 460.538,Z 517.925,A -85,B 0,C 180,E1 -8058.395,E2 -8058.395} C_VEL
LIN {X 0,Y 460.54,Z 517.93,A -85,B 0,C 180,E1 -8061.269,E2 -8061.269} C_VEL
LIN {X 0,Y 460.506,Z 517.932,A -85,B 0,C 180,E1 -8064.554,E2 -8064.554} C_VEL
LIN {X 0,Y 460.525,Z 517.927,A -85,B 0,C 180,E1 -8067.715,E2 -8067.715} C_VEL
LIN {X 0,Y 460.539,Z 517.93,A -85,B 0,C 180,E1 -8070.769,E2 -8070.769} C_VEL
LIN {X 0,Y 460.559,Z 517.922,A -85,B 0,C 180,E1 -8073.735,E2 -8073.735} C_VEL
LIN {X 0,Y 460.537,Z 517.931,A -85,B 0,C 180,E1 -8076.624,E2 -8076.624} C_VEL
LIN {X 0,Y 460.543,Z 517.927,A -85,B 0,C 180,E1 -8079.453,E2 -8079.453} C_VEL
LIN {X 0,Y 460.55,Z 517.926,A -85,B 0,C 180,E1 -8082.23,E2 -8082.23} C_VEL
LIN {X 0,Y 460.556,Z 517.93,A -85,B 0,C 180,E1 -8084.965,E2 -8084.965} C_VEL
LIN {X 0,Y 460.648,Z 517.915,A -85,B 0,C 180,E1 -8087.667,E2 -8087.667} C_VEL
LIN {X 0,Y 460.62,Z 517.923,A -85,B 0,C 180,E1 -8091.224,E2 -8091.224} C_VEL
LIN {X 0,Y 460.709,Z 517.908,A -85,B 0,C 180,E1 -8093.87,E2 -8093.87} C_VEL
LIN {X 0,Y 460.818,Z 517.897,A -85,B 0,C 180,E1 -8097.378,E2 -8097.378} C_VEL
LIN {X 0,Y 460.844,Z 517.892,A -85,B 0,C 180,E1 -8100,E2 -8100} C_VEL
LIN {X 0,Y 460.817,Z 517.898,A -85,B 0,C 180,E1 -8102.623,E2 -8102.623} C_VEL
LIN {X 0,Y 460.707,Z 518.029,A -85,B 0,C 180,E1 -8105.197,E2 -8105.197} C_VEL
LIN {X 0,Y 460.921,Z 518.983,A -85,B 0,C 180,E1 -8105.359,E2 -8105.359} C_VEL
LIN {X 0,Y 463.482,Z 526.623,A -85,B 0,C 180,E1 -8105.589,E2 -8105.589} C_VEL
LIN {X 0,Y 463.496,Z 551.36,A -85,B 0,C 180,E1 -8106.011,E2 -8106.011} C_VEL
LIN {X 0,Y 463.449,Z 564.566,A -85,B 0,C 180,E1 -8106.422,E2 -8106.422} C_VEL
LIN {X 0,Y 463.333,Z 576.446,A -85,B 0,C 180,E1 -8106.97,E2 -8106.97} C_VEL
LIN {X 0,Y 462.98,Z 588.819,A -85,B 0,C 180,E1 -8107.743,E2 -8107.743} C_VEL
LIN {X 0,Y 462.684,Z 599.738,A -85,B 0,C 180,E1 -8108.627,E2 -8108.627} C_VEL
LIN {X 0,Y 462.254,Z 609.568,A -85,B 0,C 180,E1 -8109.628,E2 -8109.628} C_VEL
LIN {X 0,Y 461.883,Z 618.424,A -85,B 0,C 180,E1 -8110.743,E2 -8110.743} C_VEL
LIN {X 0,Y 461.523,Z 625.707,A -85,B 0,C 180,E1 -8111.864,E2 -8111.864} C_VEL
LIN {X 0,Y 461.185,Z 632.799,A -85,B 0,C 180,E1 -8113.214,E2 -8113.214} C_VEL
LIN {X 0,Y 460.905,Z 638.38,A -85,B 0,C 180,E1 -8114.572,E2 -8114.572} C_VEL
LIN {X 0,Y 460.614,Z 642.911,A -85,B 0,C 180,E1 -8116.008,E2 -8116.008} C_VEL
LIN {X 0,Y 460.532,Z 644.988,A -85,B 0,C 180,E1 -8116.855,E2 -8116.855} C_VEL
LIN {X 0,Y 460.428,Z 646.756,A -85,B 0,C 180,E1 -8117.775,E2 -8117.775} C_VEL
LIN {X 0,Y 460.357,Z 648.203,A -85,B 0,C 180,E1 -8118.828,E2 -8118.828} C_VEL
LIN {X 0,Y 460.304,Z 648.924,A -85,B 0,C 180,E1 -8119.628,E2 -8119.628} C_VEL
LIN {X 0,Y 460.243,Z 649.288,A -85,B 0,C 180,E1 -8121.337,E2 -8121.337} C_VEL
LIN {X 0,Y 460.246,Z 648.745,A -85,B 0,C 180,E1 -8122.443,E2 -8122.443} C_VEL
LIN {X 0,Y 460.281,Z 647.404,A -85,B 0,C 180,E1 -8123.636,E2 -8123.636} C_VEL
LIN {X 0,Y 460.478,Z 644.245,A -85,B 0,C 180,E1 -8125.3,E2 -8125.3} C_VEL
LIN {X 0,Y 460.649,Z 640.189,A -85,B 0,C 180,E1 -8126.749,E2 -8126.749} C_VEL
LIN {X 0,Y 460.834,Z 634.724,A -85,B 0,C 180,E1 -8128.215,E2 -8128.215} C_VEL
LIN {X 0,Y 461.132,Z 628.864,A -85,B 0,C 180,E1 -8129.448,E2 -8129.448} C_VEL
LIN {X 0,Y 461.459,Z 621.657,A -85,B 0,C 180,E1 -8130.678,E2 -8130.678} C_VEL
LIN {X 0,Y 461.817,Z 613.564,A -85,B 0,C 180,E1 -8131.805,E2 -8131.805} C_VEL
LIN {X 0,Y 462.231,Z 603.663,A -85,B 0,C 180,E1 -8132.927,E2 -8132.927} C_VEL
LIN {X 0,Y 462.583,Z 594.061,A -85,B 0,C 180,E1 -8133.81,E2 -8133.81} C_VEL
LIN {X 0,Y 462.95,Z 582.377,A -85,B 0,C 180,E1 -8134.664,E2 -8134.664} C_VEL
LIN {X 0,Y 463.236,Z 570.32,A -85,B 0,C 180,E1 -8135.34,E2 -8135.34} C_VEL
LIN {X 0,Y 463.384,Z 557.549,A -85,B 0,C 180,E1 -8135.861,E2 -8135.861} C_VEL
LIN {X 0,Y 463.429,Z 544.632,A -85,B 0,C 180,E1 -8136.197,E2 -8136.197} C_VEL
LIN {X 0,Y 463.455,Z 527.224,A -85,B 0,C 180,E1 -8136.488,E2 -8136.488} C_VEL
LIN {X 0,Y 460.713,Z 519.008,A -85,B 0,C 180,E1 -8136.725,E2 -8136.725} C_VEL
LIN {X 0,Y 460.521,Z 518.029,A -85,B 0,C 180,E1 -8136.897,E2 -8136.897} C_VEL
LIN {X 0,Y 460.554,Z 517.929,A -85,B 0,C 180,E1 -8139.861,E2 -8139.861} C_VEL
LIN {X 0,Y 460.514,Z 517.933,A -85,B 0,C 180,E1 -8142.902,E2 -8142.902} C_VEL
LIN {X 0,Y 460.522,Z 517.931,A -85,B 0,C 180,E1 -8145.83,E2 -8145.83} C_VEL
LIN {X 0,Y 460.541,Z 517.929,A -85,B 0,C 180,E1 -8148.991,E2 -8148.991} C_VEL
LIN {X 0,Y 460.543,Z 517.932,A -85,B 0,C 180,E1 -8151.27,E2 -8151.27} C_VEL
LIN {X 0,Y 460.51,Z 517.929,A -85,B 0,C 180,E1 -8154.555,E2 -8154.555} C_VEL
LIN {X 0,Y 460.532,Z 517.932,A -85,B 0,C 180,E1 -8157.717,E2 -8157.717} C_VEL
LIN {X 0,Y 460.541,Z 517.926,A -85,B 0,C 180,E1 -8160.771,E2 -8160.771} C_VEL
LIN {X 0,Y 459.859,Z 518.019,A -85,B 0,C 180,E1 -8161.501,E2 -8161.501} C_VEL
LIN {X 0,Y 457.02,Z 518.364,A -85,B 0,C 180,E1 -8162.688,E2 -8162.688} C_VEL
LIN {X 0,Y 454.626,Z 518.669,A -85,B 0,C 180,E1 -8163.645,E2 -8163.645} C_VEL
LIN {X 0,Y 453.595,Z 518.792,A -85,B 0,C 180,E1 -8164.384,E2 -8164.384} C_VEL
LIN {X 0,Y 453.507,Z 518.802,A -85,B 0,C 180,E1 -8164.635,E2 -8164.635} C_VEL
LIN {X 0,Y 453.482,Z 518.809,A -85,B 0,C 180,E1 -8167.205,E2 -8167.205} C_VEL
LIN {X 0,Y 453.507,Z 518.804,A -85,B 0,C 180,E1 -8170.067,E2 -8170.067} C_VEL
LIN {X 0,Y 453.503,Z 518.803,A -85,B 0,C 180,E1 -8172.876,E2 -8172.876} C_VEL
LIN {X 0,Y 453.518,Z 518.809,A -85,B 0,C 180,E1 -8175.644,E2 -8175.644} C_VEL
LIN {X 0,Y 453.564,Z 518.795,A -85,B 0,C 180,E1 -8178.379,E2 -8178.379} C_VEL
LIN {X 0,Y 453.596,Z 518.792,A -85,B 0,C 180,E1 -8181.087,E2 -8181.087} C_VEL
LIN {X 0,Y 453.655,Z 518.791,A -85,B 0,C 180,E1 -8183.775,E2 -8183.775} C_VEL
LIN {X 0,Y 453.748,Z 518.775,A -85,B 0,C 180,E1 -8187.337,E2 -8187.337} C_VEL
LIN {X 0,Y 453.828,Z 518.767,A -85,B 0,C 180,E1 -8190,E2 -8190} C_VEL
LIN {X 0,Y 453.749,Z 518.772,A -85,B 0,C 180,E1 -8192.663,E2 -8192.663} C_VEL
LIN {X 0,Y 453.655,Z 518.786,A -85,B 0,C 180,E1 -8196.226,E2 -8196.226} C_VEL
LIN {X 0,Y 453.591,Z 518.791,A -85,B 0,C 180,E1 -8198.913,E2 -8198.913} C_VEL
LIN {X 0,Y 453.568,Z 518.795,A -85,B 0,C 180,E1 -8202.528,E2 -8202.528} C_VEL
LIN {X 0,Y 453.549,Z 518.801,A -85,B 0,C 180,E1 -8206.195,E2 -8206.195} C_VEL
LIN {X 0,Y 453.524,Z 518.8,A -85,B 0,C 180,E1 -8209.04,E2 -8209.04} C_VEL
LIN {X 0,Y 453.479,Z 518.812,A -85,B 0,C 180,E1 -8211.835,E2 -8211.835} C_VEL
LIN {X 0,Y 453.503,Z 518.803,A -85,B 0,C 180,E1 -8214.734,E2 -8214.734} C_VEL
LIN {X 0,Y 453.534,Z 518.807,A -85,B 0,C 180,E1 -8217.959,E2 -8217.959} C_VEL
LIN {X 0,Y 453.467,Z 518.809,A -85,B 0,C 180,E1 -8221.524,E2 -8221.524} C_VEL
LIN {X 0,Y 453.488,Z 518.805,A -85,B 0,C 180,E1 -8224.776,E2 -8224.776} C_VEL
LIN {X 0,Y 453.48,Z 518.81,A -85,B 0,C 180,E1 -8228.309,E2 -8228.309} C_VEL
LIN {X 0,Y 453.515,Z 518.803,A -85,B 0,C 180,E1 -8230.606,E2 -8230.606} C_VEL
LIN {X 0,Y 453.48,Z 518.805,A -85,B 0,C 180,E1 -8233.247,E2 -8233.247} C_VEL
LIN {X 0,Y 453.464,Z 518.811,A -85,B 0,C 180,E1 -8235.778,E2 -8235.778} C_VEL
LIN {X 0,Y 453.477,Z 518.813,A -85,B 0,C 180,E1 -8238.208,E2 -8238.208} C_VEL
LIN {X 0,Y 453.512,Z 518.802,A -85,B 0,C 180,E1 -8240.789,E2 -8240.789} C_VEL
LIN {X 0,Y 453.453,Z 518.813,A -85,B 0,C 180,E1 -8243.916,E2 -8243.916} C_VEL
LIN {X 0,Y 453.478,Z 518.805,A -85,B 0,C 180,E1 -8247.15,E2 -8247.15} C_VEL
LIN {X 0,Y 453.509,Z 518.81,A -85,B 0,C 180,E1 -8250.27,E2 -8250.27} C_VEL
LIN {X 0,Y 453.508,Z 518.802,A -85,B 0,C 180,E1 -8253.294,E2 -8253.294} C_VEL
LIN {X 0,Y 453.497,Z 518.811,A -85,B 0,C 180,E1 -8256.238,E2 -8256.238} C_VEL
LIN {X 0,Y 453.476,Z 518.806,A -85,B 0,C 180,E1 -8259.117,E2 -8259.117} C_VEL
LIN {X 0,Y 453.505,Z 518.805,A -85,B 0,C 180,E1 -8261.944,E2 -8261.944} C_VEL
LIN {X 0,Y 453.532,Z 518.802,A -85,B 0,C 180,E1 -8264.726,E2 -8264.726} C_VEL
LIN {X 0,Y 453.594,Z 518.791,A -85,B 0,C 180,E1 -8267.472,E2 -8267.472} C_VEL
LIN {X 0,Y 453.585,Z 518.793,A -85,B 0,C 180,E1 -8271.086,E2 -8271.086} C_VEL
LIN {X 0,Y 453.674,Z 518.782,A -85,B 0,C 180,E1 -8273.774,E2 -8273.774} C_VEL
LIN {X 0,Y 453.758,Z 518.771,A -85,B 0,C 180,E1 -8277.336,E2 -8277.336} C_VEL
LIN {X 0,Y 453.814,Z 518.766,A -85,B 0,C 180,E1 -8280,E2 -8280} C_VEL
LIN {X 0,Y 453.757,Z 518.777,A -85,B 0,C 180,E1 -8282.663,E2 -8282.663} C_VEL
LIN {X 0,Y 453.668,Z 518.786,A -85,B 0,C 180,E1 -8286.225,E2 -8286.225} C_VEL
LIN {X 0,Y 453.584,Z 518.796,A -85,B 0,C 180,E1 -8288.913,E2 -8288.913} C_VEL
LIN {X 0,Y 453.554,Z 518.804,A -85,B 0,C 180,E1 -8292.529,E2 -8292.529} C_VEL
LIN {X 0,Y 453.536,Z 518.801,A -85,B 0,C 180,E1 -8296.196,E2 -8296.196} C_VEL
LIN {X 0,Y 453.512,Z 518.804,A -85,B 0,C 180,E1 -8299.041,E2 -8299.041} C_VEL
LIN {X 0,Y 453.468,Z 518.807,A -85,B 0,C 180,E1 -8301.836,E2 -8301.836} C_VEL
LIN {X 0,Y 453.506,Z 518.81,A -85,B 0,C 180,E1 -8304.735,E2 -8304.735} C_VEL
LIN {X 0,Y 453.531,Z 518.799,A -85,B 0,C 180,E1 -8307.962,E2 -8307.962} C_VEL
LIN {X 0,Y 453.476,Z 518.814,A -85,B 0,C 180,E1 -8310.759,E2 -8310.759} C_VEL
LIN {X 0,Y 453.471,Z 518.806,A -85,B 0,C 180,E1 -8313.913,E2 -8313.913} C_VEL
LIN {X 0,Y 453.464,Z 518.81,A -85,B 0,C 180,E1 -8317.188,E2 -8317.188} C_VEL
LIN {X 0,Y 453.483,Z 518.806,A -85,B 0,C 180,E1 -8319.45,E2 -8319.45} C_VEL
LIN {X 0,Y 453.472,Z 518.806,A -85,B 0,C 180,E1 -8321.936,E2 -8321.936} C_VEL
LIN {X 0,Y 453.486,Z 518.806,A -85,B 0,C 180,E1 -8325.471,E2 -8325.471} C_VEL
LIN {X 0,Y 453.477,Z 518.806,A -85,B 0,C 180,E1 -8328.21,E2 -8328.21} C_VEL
LIN {X 0,Y 453.514,Z 518.808,A -85,B 0,C 180,E1 -8330.79,E2 -8330.79} C_VEL
LIN {X 0,Y 453.452,Z 518.811,A -85,B 0,C 180,E1 -8333.918,E2 -8333.918} C_VEL
LIN {X 0,Y 453.48,Z 518.813,A -85,B 0,C 180,E1 -8337.152,E2 -8337.152} C_VEL
LIN {X 0,Y 453.53,Z 518.871,A -85,B 0,C 180,E1 -8338.462,E2 -8338.462} C_VEL
LIN {X 0,Y 454.255,Z 522.658,A -85,B 0,C 180,E1 -8339.3,E2 -8339.3} C_VEL
LIN {X 0,Y 456.465,Z 533.539,A -85,B 0,C 180,E1 -8341.492,E2 -8341.492} C_VEL
LIN {X 0,Y 456.327,Z 540.146,A -85,B 0,C 180,E1 -8342.728,E2 -8342.728} C_VEL
LIN {X 0,Y 455.342,Z 558.722,A -85,B 0,C 180,E1 -8346.122,E2 -8346.122} C_VEL
LIN {X 0,Y 454.503,Z 577.034,A -85,B 0,C 180,E1 -8349.404,E2 -8349.404} C_VEL
LIN {X 0,Y 453.824,Z 595.457,A -85,B 0,C 180,E1 -8352.656,E2 -8352.656} C_VEL
LIN {X 0,Y 453.371,Z 612.529,A -85,B 0,C 180,E1 -8355.64,E2 -8355.64} C_VEL
LIN {X 0,Y 453.321,Z 614.372,A -85,B 0,C 180,E1 -8355.925,E2 -8355.925} C_VEL
LIN {X 0,Y 455.726,Z 642.371,A -85,B 0,C 180,E1 -8356.524,E2 -8356.524} C_VEL
LIN {X 0,Y 455.212,Z 696.03,A -85,B 0,C 180,E1 -8357.495,E2 -8357.495} C_VEL
LIN {X 0,Y 454.791,Z 708.331,A -85,B 0,C 180,E1 -8357.902,E2 -8357.902} C_VEL
LIN {X 0,Y 454.368,Z 720.427,A -85,B 0,C 180,E1 -8358.513,E2 -8358.513} C_VEL
LIN {X 0,Y 453.862,Z 731.568,A -85,B 0,C 180,E1 -8359.291,E2 -8359.291} C_VEL
LIN {X 0,Y 453.457,Z 741.376,A -85,B 0,C 180,E1 -8360.184,E2 -8360.184} C_VEL
LIN {X 0,Y 453.136,Z 749.24,A -85,B 0,C 180,E1 -8361.078,E2 -8361.078} C_VEL
LIN {X 0,Y 452.953,Z 757.16,A -85,B 0,C 180,E1 -8362.197,E2 -8362.197} C_VEL
LIN {X 0,Y 452.851,Z 764.529,A -85,B 0,C 180,E1 -8363.529,E2 -8363.529} C_VEL
LIN {X 0,Y 452.769,Z 769.337,A -85,B 0,C 180,E1 -8364.656,E2 -8364.656} C_VEL
LIN {X 0,Y 452.904,Z 773.689,A -85,B 0,C 180,E1 -8365.996,E2 -8365.996} C_VEL
LIN {X 0,Y 452.839,Z 776.633,A -85,B 0,C 180,E1 -8367.331,E2 -8367.331} C_VEL
LIN {X 0,Y 452.834,Z 777.906,A -85,B 0,C 180,E1 -8368.221,E2 -8368.221} C_VEL
LIN {X 0,Y 452.848,Z 778.634,A -85,B 0,C 180,E1 -8369.111,E2 -8369.111} C_VEL
LIN {X 0,Y 453.013,Z 778.879,A -85,B 0,C 180,E1 -8370,E2 -8370} C_VEL
LIN {X 0,Y 452.863,Z 778.519,A -85,B 0,C 180,E1 -8370.889,E2 -8370.889} C_VEL
LIN {X 0,Y 452.861,Z 777.689,A -85,B 0,C 180,E1 -8371.779,E2 -8371.779} C_VEL
LIN {X 0,Y 452.873,Z 776.291,A -85,B 0,C 180,E1 -8372.668,E2 -8372.668} C_VEL
LIN {X 0,Y 452.918,Z 773.181,A -85,B 0,C 180,E1 -8374.004,E2 -8374.004} C_VEL
LIN {X 0,Y 452.835,Z 768.641,A -85,B 0,C 180,E1 -8375.343,E2 -8375.343} C_VEL
LIN {X 0,Y 452.909,Z 763.695,A -85,B 0,C 180,E1 -8376.463,E2 -8376.463} C_VEL
LIN {X 0,Y 452.953,Z 757.513,A -85,B 0,C 180,E1 -8377.578,E2 -8377.578} C_VEL
LIN {X 0,Y 453.113,Z 749.738,A -85,B 0,C 180,E1 -8378.698,E2 -8378.698} C_VEL
LIN {X 0,Y 453.397,Z 741.047,A -85,B 0,C 180,E1 -8379.704,E2 -8379.704} C_VEL
LIN {X 0,Y 453.755,Z 731.331,A -85,B 0,C 180,E1 -8380.598,E2 -8380.598} C_VEL
LIN {X 0,Y 454.222,Z 720.417,A -85,B 0,C 180,E1 -8381.377,E2 -8381.377} C_VEL
LIN {X 0,Y 454.659,Z 708.979,A -85,B 0,C 180,E1 -8381.988,E2 -8381.988} C_VEL
LIN {X 0,Y 455.164,Z 696.007,A -85,B 0,C 180,E1 -8382.455,E2 -8382.455} C_VEL
LIN {X 0,Y 455.351,Z 680.196,A -85,B 0,C 180,E1 -8382.773,E2 -8382.773} C_VEL
LIN {X 0,Y 455.443,Z 638.552,A -85,B 0,C 180,E1 -8383.499,E2 -8383.499} C_VEL
LIN {X 0,Y 453.303,Z 609.986,A -85,B 0,C 180,E1 -8384.105,E2 -8384.105} C_VEL
LIN {X 0,Y 453.384,Z 602.728,A -85,B 0,C 180,E1 -8385.279,E2 -8385.279} C_VEL
LIN {X 0,Y 453.72,Z 585.104,A -85,B 0,C 180,E1 -8388.28,E2 -8388.28} C_VEL
LIN {X 0,Y 454.266,Z 566.189,A -85,B 0,C 180,E1 -8391.557,E2 -8391.557} C_VEL
LIN {X 0,Y 454.887,Z 548.759,A -85,B 0,C 180,E1 -8394.654,E2 -8394.654} C_VEL
LIN {X 0,Y 455.594,Z 531.579,A -85,B 0,C 180,E1 -8397.808,E2 -8397.808} C_VEL
LIN {X 0,Y 454.718,Z 524.858,A -85,B 0,C 180,E1 -8399.133,E2 -8399.133} C_VEL
LIN {X 0,Y 453.54,Z 518.923,A -85,B 0,C 180,E1 -8400.398,E2 -8400.398} C_VEL
LIN {X 0,Y 453.474,Z 518.811,A -85,B 0,C 180,E1 -8403.912,E2 -8403.912} C_VEL
LIN {X 0,Y 453.466,Z 518.815,A -85,B 0,C 180,E1 -8407.187,E2 -8407.187} C_VEL
LIN {X 0,Y 453.5,Z 518.806,A -85,B 0,C 180,E1 -8409.447,E2 -8409.447} C_VEL
LIN {X 0,Y 453.465,Z 518.814,A -85,B 0,C 180,E1 -8412.993,E2 -8412.993} C_VEL
LIN {X 0,Y 453.471,Z 518.808,A -85,B 0,C 180,E1 -8415.78,E2 -8415.78} C_VEL
LIN {X 0,Y 453.489,Z 518.802,A -85,B 0,C 180,E1 -8418.211,E2 -8418.211} C_VEL
LIN {X 0,Y 453.526,Z 518.804,A -85,B 0,C 180,E1 -8420.787,E2 -8420.787} C_VEL
LIN {X 0,Y 453.45,Z 518.808,A -85,B 0,C 180,E1 -8423.917,E2 -8423.917} C_VEL
LIN {X 0,Y 453.475,Z 518.808,A -85,B 0,C 180,E1 -8427.151,E2 -8427.151} C_VEL
LIN {X 0,Y 453.506,Z 518.804,A -85,B 0,C 180,E1 -8430.271,E2 -8430.271} C_VEL
LIN {X 0,Y 453.505,Z 518.803,A -85,B 0,C 180,E1 -8433.294,E2 -8433.294} C_VEL
LIN {X 0,Y 453.494,Z 518.806,A -85,B 0,C 180,E1 -8436.239,E2 -8436.239} C_VEL
LIN {X 0,Y 453.474,Z 518.809,A -85,B 0,C 180,E1 -8439.117,E2 -8439.117} C_VEL
LIN {X 0,Y 453.502,Z 518.803,A -85,B 0,C 180,E1 -8441.944,E2 -8441.944} C_VEL
LIN {X 0,Y 453.53,Z 518.804,A -85,B 0,C 180,E1 -8444.726,E2 -8444.726} C_VEL
LIN {X 0,Y 453.592,Z 518.795,A -85,B 0,C 180,E1 -8447.472,E2 -8447.472} C_VEL
LIN {X 0,Y 453.584,Z 518.799,A -85,B 0,C 180,E1 -8451.087,E2 -8451.087} C_VEL
LIN {X 0,Y 453.675,Z 518.785,A -85,B 0,C 180,E1 -8453.775,E2 -8453.775} C_VEL
LIN {X 0,Y 453.758,Z 518.776,A -85,B 0,C 180,E1 -8457.337,E2 -8457.337} C_VEL
LIN {X 0,Y 453.814,Z 518.768,A -85,B 0,C 180,E1 -8460,E2 -8460} C_VEL
LIN {X 0,Y 453.758,Z 518.777,A -85,B 0,C 180,E1 -8462.664,E2 -8462.664} C_VEL
LIN {X 0,Y 453.635,Z 518.902,A -85,B 0,C 180,E1 -8464.944,E2 -8464.944} C_VEL
LIN {X 0,Y 453.84,Z 519.824,A -85,B 0,C 180,E1 -8465.109,E2 -8465.109} C_VEL
LIN {X 0,Y 456.625,Z 527.963,A -85,B 0,C 180,E1 -8465.368,E2 -8465.368} C_VEL
LIN {X 0,Y 456.685,Z 551.559,A -85,B 0,C 180,E1 -8465.769,E2 -8465.769} C_VEL
LIN {X 0,Y 456.63,Z 565.11,A -85,B 0,C 180,E1 -8466.185,E2 -8466.185} C_VEL
LIN {X 0,Y 456.536,Z 577.186,A -85,B 0,C 180,E1 -8466.741,E2 -8466.741} C_VEL
LIN {X 0,Y 456.259,Z 588.059,A -85,B 0,C 180,E1 -8467.412,E2 -8467.412} C_VEL
LIN {X 0,Y 455.874,Z 599.374,A -85,B 0,C 180,E1 -8468.31,E2 -8468.31} C_VEL
LIN {X 0,Y 455.481,Z 609.11,A -85,B 0,C 180,E1 -8469.279,E2 -8469.279} C_VEL
LIN {X 0,Y 455.034,Z 618.566,A -85,B 0,C 180,E1 -8470.456,E2 -8470.456} C_VEL
LIN {X 0,Y 454.558,Z 627.349,A -85,B 0,C 180,E1 -8471.822,E2 -8471.822} C_VEL
LIN {X 0,Y 454.229,Z 634.218,A -85,B 0,C 180,E1 -8473.179,E2 -8473.179} C_VEL
LIN {X 0,Y 453.956,Z 638.978,A -85,B 0,C 180,E1 -8474.342,E2 -8474.342} C_VEL
LIN {X 0,Y 453.68,Z 643.362,A -85,B 0,C 180,E1 -8475.707,E2 -8475.707} C_VEL
LIN {X 0,Y 453.482,Z 646.716,A -85,B 0,C 180,E1 -8477.126,E2 -8477.126} C_VEL
LIN {X 0,Y 453.391,Z 648.313,A -85,B 0,C 180,E1 -8478.061,E2 -8478.061} C_VEL
LIN {X 0,Y 453.34,Z 649.46,A -85,B 0,C 180,E1 -8479,E2 -8479} C_VEL
LIN {X 0,Y 453.253,Z 650.126,A -85,B 0,C 180,E1 -8479.946,E2 -8479.946} C_VEL
LIN {X 0,Y 453.21,Z 650.258,A -85,B 0,C 180,E1 -8481.502,E2 -8481.502} C_VEL
LIN {X 0,Y 453.227,Z 649.411,A -85,B 0,C 180,E1 -8482.81,E2 -8482.81} C_VEL
LIN {X 0,Y 453.276,Z 648.168,A -85,B 0,C 180,E1 -8483.828,E2 -8483.828} C_VEL
LIN {X 0,Y 453.445,Z 645.518,A -85,B 0,C 180,E1 -8485.229,E2 -8485.229} C_VEL
LIN {X 0,Y 453.65,Z 641.544,A -85,B 0,C 180,E1 -8486.697,E2 -8486.697} C_VEL
LIN {X 0,Y 453.849,Z 635.673,A -85,B 0,C 180,E1 -8488.307,E2 -8488.307} C_VEL
LIN {X 0,Y 454.174,Z 629.141,A -85,B 0,C 180,E1 -8489.682,E2 -8489.682} C_VEL
LIN {X 0,Y 454.568,Z 621.7,A -85,B 0,C 180,E1 -8490.936,E2 -8490.936} C_VEL
LIN {X 0,Y 454.999,Z 612.394,A -85,B 0,C 180,E1 -8492.207,E2 -8492.207} C_VEL
LIN {X 0,Y 455.369,Z 603.224,A -85,B 0,C 180,E1 -8493.221,E2 -8493.221} C_VEL
LIN {X 0,Y 455.746,Z 593.191,A -85,B 0,C 180,E1 -8494.121,E2 -8494.121} C_VEL
LIN {X 0,Y 456.098,Z 581.766,A -85,B 0,C 180,E1 -8494.938,E2 -8494.938} C_VEL
LIN {X 0,Y 456.365,Z 570.326,A -85,B 0,C 180,E1 -8495.57,E2 -8495.57} C_VEL
LIN {X 0,Y 456.504,Z 557.35,A -85,B 0,C 180,E1 -8496.086,E2 -8496.086} C_VEL
LIN {X 0,Y 456.541,Z 544.094,A -85,B 0,C 180,E1 -8496.42,E2 -8496.42} C_VEL
LIN {X 0,Y 456.414,Z 528.143,A -85,B 0,C 180,E1 -8496.69,E2 -8496.69} C_VEL
LIN {X 0,Y 453.668,Z 519.855,A -85,B 0,C 180,E1 -8496.939,E2 -8496.939} C_VEL
LIN {X 0,Y 453.509,Z 518.931,A -85,B 0,C 180,E1 -8497.096,E2 -8497.096} C_VEL
LIN {X 0,Y 453.513,Z 518.809,A -85,B 0,C 180,E1 -8499.448,E2 -8499.448} C_VEL
LIN {X 0,Y 453.465,Z 518.812,A -85,B 0,C 180,E1 -8502.995,E2 -8502.995} C_VEL
LIN {X 0,Y 453.475,Z 518.809,A -85,B 0,C 180,E1 -8505.781,E2 -8505.781} C_VEL
LIN {X 0,Y 453.494,Z 518.804,A -85,B 0,C 180,E1 -8508.212,E2 -8508.212} C_VEL
LIN {X 0,Y 453.529,Z 518.8,A -85,B 0,C 180,E1 -8510.789,E2 -8510.789} C_VEL
LIN {X 0,Y 453.453,Z 518.811,A -85,B 0,C 180,E1 -8513.918,E2 -8513.918} C_VEL
LIN {X 0,Y 453.483,Z 518.809,A -85,B 0,C 180,E1 -8517.152,E2 -8517.152} C_VEL
LIN {X 0,Y 453.476,Z 518.806,A -85,B 0,C 180,E1 -8520.269,E2 -8520.269} C_VEL
LIN {X 0,Y 453.512,Z 518.806,A -85,B 0,C 180,E1 -8523.295,E2 -8523.295} C_VEL
LIN {X 0,Y 453.507,Z 518.802,A -85,B 0,C 180,E1 -8524.635,E2 -8524.635} C_VEL
LIN {X 0,Y 452.828,Z 518.892,A -85,B 0,C 180,E1 -8525.375,E2 -8525.375} C_VEL
LIN {X 0,Y 449.962,Z 519.245,A -85,B 0,C 180,E1 -8526.578,E2 -8526.578} C_VEL
LIN {X 0,Y 447.551,Z 519.552,A -85,B 0,C 180,E1 -8527.549,E2 -8527.549} C_VEL
LIN {X 0,Y 446.527,Z 519.673,A -85,B 0,C 180,E1 -8528.299,E2 -8528.299} C_VEL
LIN {X 0,Y 446.449,Z 519.681,A -85,B 0,C 180,E1 -8528.553,E2 -8528.553} C_VEL
LIN {X 0,Y 446.456,Z 519.688,A -85,B 0,C 180,E1 -8531.65,E2 -8531.65} C_VEL
LIN {X 0,Y 446.512,Z 519.673,A -85,B 0,C 180,E1 -8534.48,E2 -8534.48} C_VEL
LIN {X 0,Y 446.522,Z 519.674,A -85,B 0,C 180,E1 -8538.194,E2 -8538.194} C_VEL
LIN {X 0,Y 446.541,Z 519.67,A -85,B 0,C 180,E1 -8540.945,E2 -8540.945} C_VEL
LIN {X 0,Y 446.623,Z 519.668,A -85,B 0,C 180,E1 -8543.676,E2 -8543.676} C_VEL
LIN {X 0,Y 446.695,Z 519.653,A -85,B 0,C 180,E1 -8547.295,E2 -8547.295} C_VEL
LIN {X 0,Y 446.798,Z 519.642,A -85,B 0,C 180,E1 -8550,E2 -8550} C_VEL
LIN {X 0,Y 446.696,Z 519.65,A -85,B 0,C 180,E1 -8552.705,E2 -8552.705} C_VEL
LIN {X 0,Y 446.624,Z 519.661,A -85,B 0,C 180,E1 -8556.324,E2 -8556.324} C_VEL
LIN {X 0,Y 446.528,Z 519.677,A -85,B 0,C 180,E1 -8559.97,E2 -8559.97} C_VEL
LIN {X 0,Y 446.526,Z 519.672,A -85,B 0,C 180,E1 -8562.729,E2 -8562.729} C_VEL
LIN {X 0,Y 446.5,Z 519.678,A -85,B 0,C 180,E1 -8566.227,E2 -8566.227} C_VEL
LIN {X 0,Y 446.473,Z 519.679,A -85,B 0,C 180,E1 -8569.303,E2 -8569.303} C_VEL
LIN {X 0,Y 446.421,Z 519.689,A -85,B 0,C 180,E1 -8572.199,E2 -8572.199} C_VEL
LIN {X 0,Y 446.447,Z 519.682,A -85,B 0,C 180,E1 -8575.152,E2 -8575.152} C_VEL
LIN {X 0,Y 446.487,Z 519.682,A -85,B 0,C 180,E1 -8578.178,E2 -8578.178} C_VEL
LIN {X 0,Y 446.42,Z 519.69,A -85,B 0,C 180,E1 -8581.774,E2 -8581.774} C_VEL
LIN {X 0,Y 446.429,Z 519.686,A -85,B 0,C 180,E1 -8584.522,E2 -8584.522} C_VEL
LIN {X 0,Y 446.435,Z 519.691,A -85,B 0,C 180,E1 -8588.082,E2 -8588.082} C_VEL
LIN {X 0,Y 446.446,Z 519.682,A -85,B 0,C 180,E1 -8590.92,E2 -8590.92} C_VEL
LIN {X 0,Y 446.444,Z 519.686,A -85,B 0,C 180,E1 -8593.84,E2 -8593.84} C_VEL
LIN {X 0,Y 446.397,Z 519.692,A -85,B 0,C 180,E1 -8596.402,E2 -8596.402} C_VEL
LIN {X 0,Y 446.424,Z 519.684,A -85,B 0,C 180,E1 -8599.081,E2 -8599.081} C_VEL
LIN {X 0,Y 446.427,Z 519.689,A -85,B 0,C 180,E1 -8601.917,E2 -8601.917} C_VEL
LIN {X 0,Y 446.426,Z 519.685,A -85,B 0,C 180,E1 -8605.476,E2 -8605.476} C_VEL
LIN {X 0,Y 446.426,Z 519.686,A -85,B 0,C 180,E1 -8608.7,E2 -8608.7} C_VEL
LIN {X 0,Y 446.479,Z 519.68,A -85,B 0,C 180,E1 -8611.821,E2 -8611.821} C_VEL
LIN {X 0,Y 446.452,Z 519.682,A -85,B 0,C 180,E1 -8614.847,E2 -8614.847} C_VEL
LIN {X 0,Y 446.441,Z 519.69,A -85,B 0,C 180,E1 -8618.244,E2 -8618.244} C_VEL
LIN {X 0,Y 446.45,Z 519.682,A -85,B 0,C 180,E1 -8621.649,E2 -8621.649} C_VEL
LIN {X 0,Y 446.5,Z 519.681,A -85,B 0,C 180,E1 -8624.479,E2 -8624.479} C_VEL
LIN {X 0,Y 446.531,Z 519.676,A -85,B 0,C 180,E1 -8628.193,E2 -8628.193} C_VEL
LIN {X 0,Y 446.592,Z 519.665,A -85,B 0,C 180,E1 -8631.857,E2 -8631.857} C_VEL
LIN {X 0,Y 446.644,Z 519.663,A -85,B 0,C 180,E1 -8634.582,E2 -8634.582} C_VEL
LIN {X 0,Y 446.702,Z 519.65,A -85,B 0,C 180,E1 -8637.294,E2 -8637.294} C_VEL
LIN {X 0,Y 446.784,Z 519.641,A -85,B 0,C 180,E1 -8640,E2 -8640} C_VEL
LIN {X 0,Y 446.701,Z 519.655,A -85,B 0,C 180,E1 -8642.705,E2 -8642.705} C_VEL
LIN {X 0,Y 446.638,Z 519.663,A -85,B 0,C 180,E1 -8646.324,E2 -8646.324} C_VEL
LIN {X 0,Y 446.529,Z 519.673,A -85,B 0,C 180,E1 -8649.055,E2 -8649.055} C_VEL
LIN {X 0,Y 446.512,Z 519.679,A -85,B 0,C 180,E1 -8652.73,E2 -8652.73} C_VEL
LIN {X 0,Y 446.487,Z 519.679,A -85,B 0,C 180,E1 -8656.228,E2 -8656.228} C_VEL
LIN {X 0,Y 446.461,Z 519.68,A -85,B 0,C 180,E1 -8659.303,E2 -8659.303} C_VEL
LIN {X 0,Y 446.41,Z 519.688,A -85,B 0,C 180,E1 -8662.2,E2 -8662.2} C_VEL
LIN {X 0,Y 446.45,Z 519.683,A -85,B 0,C 180,E1 -8665.152,E2 -8665.152} C_VEL
LIN {X 0,Y 446.477,Z 519.679,A -85,B 0,C 180,E1 -8668.179,E2 -8668.179} C_VEL
LIN {X 0,Y 446.412,Z 519.687,A -85,B 0,C 180,E1 -8671.3,E2 -8671.3} C_VEL
LIN {X 0,Y 446.423,Z 519.689,A -85,B 0,C 180,E1 -8674.523,E2 -8674.523} C_VEL
LIN {X 0,Y 446.424,Z 519.685,A -85,B 0,C 180,E1 -8678.082,E2 -8678.082} C_VEL
LIN {X 0,Y 446.422,Z 519.691,A -85,B 0,C 180,E1 -8680.918,E2 -8680.918} C_VEL
LIN {X 0,Y 446.418,Z 519.685,A -85,B 0,C 180,E1 -8683.844,E2 -8683.844} C_VEL
LIN {X 0,Y 446.416,Z 519.688,A -85,B 0,C 180,E1 -8686.401,E2 -8686.401} C_VEL
LIN {X 0,Y 446.447,Z 519.681,A -85,B 0,C 180,E1 -8689.804,E2 -8689.804} C_VEL
LIN {X 0,Y 446.425,Z 519.684,A -85,B 0,C 180,E1 -8692.124,E2 -8692.124} C_VEL
LIN {X 0,Y 446.426,Z 519.69,A -85,B 0,C 180,E1 -8695.478,E2 -8695.478} C_VEL
LIN {X 0,Y 446.533,Z 519.821,A -85,B 0,C 180,E1 -8698.295,E2 -8698.295} C_VEL
LIN {X 0,Y 449.27,Z 533.585,A -85,B 0,C 180,E1 -8701.165,E2 -8701.165} C_VEL
LIN {X 0,Y 449.549,Z 538.006,A -85,B 0,C 180,E1 -8702.031,E2 -8702.031} C_VEL
LIN {X 0,Y 448.442,Z 557.405,A -85,B 0,C 180,E1 -8705.65,E2 -8705.65} C_VEL
LIN {X 0,Y 447.474,Z 577.404,A -85,B 0,C 180,E1 -8709.306,E2 -8709.306} C_VEL
LIN {X 0,Y 446.784,Z 594.438,A -85,B 0,C 180,E1 -8712.374,E2 -8712.374} C_VEL
LIN {X 0,Y 446.288,Z 612.854,A -85,B 0,C 180,E1 -8715.64,E2 -8715.64} C_VEL
LIN {X 0,Y 446.374,Z 614.902,A -85,B 0,C 180,E1 -8715.745,E2 -8715.745} C_VEL
LIN {X 0,Y 448.803,Z 642.527,A -85,B 0,C 180,E1 -8716.329,E2 -8716.329} C_VEL
LIN {X 0,Y 448.289,Z 694.814,A -85,B 0,C 180,E1 -8717.299,E2 -8717.299} C_VEL
LIN {X 0,Y 447.889,Z 705.785,A -85,B 0,C 180,E1 -8717.655,E2 -8717.655} C_VEL
LIN {X 0,Y 447.435,Z 717.328,A -85,B 0,C 180,E1 -8718.218,E2 -8718.218} C_VEL
LIN {X 0,Y 446.966,Z 727.59,A -85,B 0,C 180,E1 -8718.895,E2 -8718.895} C_VEL
LIN {X 0,Y 446.503,Z 738.059,A -85,B 0,C 180,E1 -8719.801,E2 -8719.801} C_VEL
LIN {X 0,Y 446.184,Z 746.369,A -85,B 0,C 180,E1 -8720.709,E2 -8720.709} C_VEL
LIN {X 0,Y 445.94,Z 754.675,A -85,B 0,C 180,E1 -8721.846,E2 -8721.846} C_VEL
LIN {X 0,Y 445.814,Z 761.458,A -85,B 0,C 180,E1 -8723.016,E2 -8723.016} C_VEL
LIN {X 0,Y 445.79,Z 766.547,A -85,B 0,C 180,E1 -8724.118,E2 -8724.118} C_VEL
LIN {X 0,Y 445.783,Z 771.398,A -85,B 0,C 180,E1 -8725.479,E2 -8725.479} C_VEL
LIN {X 0,Y 445.855,Z 773.807,A -85,B 0,C 180,E1 -8726.385,E2 -8726.385} C_VEL
LIN {X 0,Y 445.795,Z 775.636,A -85,B 0,C 180,E1 -8727.289,E2 -8727.289} C_VEL
LIN {X 0,Y 445.795,Z 776.909,A -85,B 0,C 180,E1 -8728.193,E2 -8728.193} C_VEL
LIN {X 0,Y 445.814,Z 777.641,A -85,B 0,C 180,E1 -8729.097,E2 -8729.097} C_VEL
LIN {X 0,Y 445.992,Z 777.884,A -85,B 0,C 180,E1 -8730,E2 -8730} C_VEL
LIN {X 0,Y 445.829,Z 777.521,A -85,B 0,C 180,E1 -8730.903,E2 -8730.903} C_VEL
LIN {X 0,Y 445.822,Z 776.686,A -85,B 0,C 180,E1 -8731.807,E2 -8731.807} C_VEL
LIN {X 0,Y 445.828,Z 775.278,A -85,B 0,C 180,E1 -8732.71,E2 -8732.71} C_VEL
LIN {X 0,Y 445.873,Z 772.16,A -85,B 0,C 180,E1 -8734.067,E2 -8734.067} C_VEL
LIN {X 0,Y 445.775,Z 767.609,A -85,B 0,C 180,E1 -8735.428,E2 -8735.428} C_VEL
LIN {X 0,Y 445.822,Z 761.926,A -85,B 0,C 180,E1 -8736.716,E2 -8736.716} C_VEL
LIN {X 0,Y 445.909,Z 755.047,A -85,B 0,C 180,E1 -8737.927,E2 -8737.927} C_VEL
LIN {X 0,Y 446.082,Z 746.951,A -85,B 0,C 180,E1 -8739.064,E2 -8739.064} C_VEL
LIN {X 0,Y 446.41,Z 737.791,A -85,B 0,C 180,E1 -8740.087,E2 -8740.087} C_VEL
LIN {X 0,Y 446.859,Z 727.498,A -85,B 0,C 180,E1 -8740.993,E2 -8740.993} C_VEL
LIN {X 0,Y 447.3,Z 717.647,A -85,B 0,C 180,E1 -8741.671,E2 -8741.671} C_VEL
LIN {X 0,Y 447.76,Z 706.833,A -85,B 0,C 180,E1 -8742.233,E2 -8742.233} C_VEL
LIN {X 0,Y 448.224,Z 694.389,A -85,B 0,C 180,E1 -8742.68,E2 -8742.68} C_VEL
LIN {X 0,Y 448.461,Z 676.745,A -85,B 0,C 180,E1 -8743.032,E2 -8743.032} C_VEL
LIN {X 0,Y 448.611,Z 639.568,A -85,B 0,C 180,E1 -8743.696,E2 -8743.696} C_VEL
LIN {X 0,Y 446.272,Z 608.507,A -85,B 0,C 180,E1 -8744.37,E2 -8744.37} C_VEL
LIN {X 0,Y 446.305,Z 605.476,A -85,B 0,C 180,E1 -8744.826,E2 -8744.826} C_VEL
LIN {X 0,Y 446.619,Z 586.55,A -85,B 0,C 180,E1 -8748.106,E2 -8748.106} C_VEL
LIN {X 0,Y 447.176,Z 567.78,A -85,B 0,C 180,E1 -8751.422,E2 -8751.422} C_VEL
LIN {X 0,Y 447.846,Z 549.658,A -85,B 0,C 180,E1 -8754.705,E2 -8754.705} C_VEL
LIN {X 0,Y 448.591,Z 533.245,A -85,B 0,C 180,E1 -8757.78,E2 -8757.78} C_VEL
LIN {X 0,Y 448.078,Z 528.172,A -85,B 0,C 180,E1 -8758.791,E2 -8758.791} C_VEL
LIN {X 0,Y 446.504,Z 519.764,A -85,B 0,C 180,E1 -8760.602,E2 -8760.602} C_VEL
LIN {X 0,Y 446.441,Z 519.689,A -85,B 0,C 180,E1 -8763.453,E2 -8763.453} C_VEL
LIN {X 0,Y 446.404,Z 519.694,A -85,B 0,C 180,E1 -8766.744,E2 -8766.744} C_VEL
LIN {X 0,Y 446.463,Z 519.682,A -85,B 0,C 180,E1 -8769.527,E2 -8769.527} C_VEL
LIN {X 0,Y 446.428,Z 519.687,A -85,B 0,C 180,E1 -8772.603,E2 -8772.603} C_VEL
LIN {X 0,Y 446.452,Z 519.685,A -85,B 0,C 180,E1 -8775.102,E2 -8775.102} C_VEL
LIN {X 0,Y 446.437,Z 519.684,A -85,B 0,C 180,E1 -8778.61,E2 -8778.61} C_VEL
LIN {X 0,Y 446.469,Z 519.682,A -85,B 0,C 180,E1 -8780.976,E2 -8780.976} C_VEL
LIN {X 0,Y 446.414,Z 519.686,A -85,B 0,C 180,E1 -8784.374,E2 -8784.374} C_VEL
LIN {X 0,Y 446.422,Z 519.685,A -85,B 0,C 180,E1 -8787.639,E2 -8787.639} C_VEL
LIN {X 0,Y 446.461,Z 519.683,A -85,B 0,C 180,E1 -8790.792,E2 -8790.792} C_VEL
LIN {X 0,Y 446.469,Z 519.677,A -85,B 0,C 180,E1 -8793.848,E2 -8793.848} C_VEL
LIN {X 0,Y 446.42,Z 519.689,A -85,B 0,C 180,E1 -8796.823,E2 -8796.823} C_VEL
LIN {X 0,Y 446.435,Z 519.683,A -85,B 0,C 180,E1 -8799.737,E2 -8799.737} C_VEL
LIN {X 0,Y 446.454,Z 519.684,A -85,B 0,C 180,E1 -8802.597,E2 -8802.597} C_VEL
LIN {X 0,Y 446.463,Z 519.684,A -85,B 0,C 180,E1 -8805.412,E2 -8805.412} C_VEL
LIN {X 0,Y 446.536,Z 519.674,A -85,B 0,C 180,E1 -8808.194,E2 -8808.194} C_VEL
LIN {X 0,Y 446.591,Z 519.667,A -85,B 0,C 180,E1 -8811.858,E2 -8811.858} C_VEL
LIN {X 0,Y 446.644,Z 519.663,A -85,B 0,C 180,E1 -8814.583,E2 -8814.583} C_VEL
LIN {X 0,Y 446.702,Z 519.656,A -85,B 0,C 180,E1 -8817.295,E2 -8817.295} C_VEL
LIN {X 0,Y 446.785,Z 519.644,A -85,B 0,C 180,E1 -8820,E2 -8820} C_VEL
LIN {X 0,Y 446.702,Z 519.656,A -85,B 0,C 180,E1 -8822.706,E2 -8822.706} C_VEL
LIN {X 0,Y 446.533,Z 519.785,A -85,B 0,C 180,E1 -8824.684,E2 -8824.684} C_VEL
LIN {X 0,Y 446.73,Z 520.695,A -85,B 0,C 180,E1 -8824.851,E2 -8824.851} C_VEL
LIN {X 0,Y 449.87,Z 529.489,A -85,B 0,C 180,E1 -8825.138,E2 -8825.138} C_VEL
LIN {X 0,Y 449.89,Z 553.956,A -85,B 0,C 180,E1 -8825.575,E2 -8825.575} C_VEL
LIN {X 0,Y 449.829,Z 567.115,A -85,B 0,C 180,E1 -8825.998,E2 -8825.998} C_VEL
LIN {X 0,Y 449.681,Z 578.96,A -85,B 0,C 180,E1 -8826.563,E2 -8826.563} C_VEL
LIN {X 0,Y 449.33,Z 590.517,A -85,B 0,C 180,E1 -8827.301,E2 -8827.301} C_VEL
LIN {X 0,Y 449.013,Z 601.524,A -85,B 0,C 180,E1 -8828.21,E2 -8828.21} C_VEL
LIN {X 0,Y 448.564,Z 611.375,A -85,B 0,C 180,E1 -8829.233,E2 -8829.233} C_VEL
LIN {X 0,Y 448.127,Z 620.358,A -85,B 0,C 180,E1 -8830.391,E2 -8830.391} C_VEL
LIN {X 0,Y 447.709,Z 627.68,A -85,B 0,C 180,E1 -8831.546,E2 -8831.546} C_VEL
LIN {X 0,Y 447.385,Z 633.705,A -85,B 0,C 180,E1 -8832.705,E2 -8832.705} C_VEL
LIN {X 0,Y 447.025,Z 639.581,A -85,B 0,C 180,E1 -8834.105,E2 -8834.105} C_VEL
LIN {X 0,Y 446.714,Z 644.146,A -85,B 0,C 180,E1 -8835.513,E2 -8835.513} C_VEL
LIN {X 0,Y 446.562,Z 646.503,A -85,B 0,C 180,E1 -8836.457,E2 -8836.457} C_VEL
LIN {X 0,Y 446.439,Z 648.409,A -85,B 0,C 180,E1 -8837.404,E2 -8837.404} C_VEL
LIN {X 0,Y 446.316,Z 650.625,A -85,B 0,C 180,E1 -8839.13,E2 -8839.13} C_VEL
LIN {X 0,Y 446.212,Z 651.306,A -85,B 0,C 180,E1 -8840.274,E2 -8840.274} C_VEL
LIN {X 0,Y 446.185,Z 651.225,A -85,B 0,C 180,E1 -8841.673,E2 -8841.673} C_VEL
LIN {X 0,Y 446.24,Z 650.042,A -85,B 0,C 180,E1 -8843.187,E2 -8843.187} C_VEL
LIN {X 0,Y 446.303,Z 648.643,A -85,B 0,C 180,E1 -8844.169,E2 -8844.169} C_VEL
LIN {X 0,Y 446.497,Z 645.609,A -85,B 0,C 180,E1 -8845.65,E2 -8845.65} C_VEL
LIN {X 0,Y 446.697,Z 641.313,A -85,B 0,C 180,E1 -8847.147,E2 -8847.147} C_VEL
LIN {X 0,Y 446.949,Z 635.486,A -85,B 0,C 180,E1 -8848.664,E2 -8848.664} C_VEL
LIN {X 0,Y 447.35,Z 627.977,A -85,B 0,C 180,E1 -8850.181,E2 -8850.181} C_VEL
LIN {X 0,Y 447.773,Z 620.017,A -85,B 0,C 180,E1 -8851.459,E2 -8851.459} C_VEL
LIN {X 0,Y 448.187,Z 611.099,A -85,B 0,C 180,E1 -8852.618,E2 -8852.618} C_VEL
LIN {X 0,Y 448.551,Z 601.355,A -85,B 0,C 180,E1 -8853.653,E2 -8853.653} C_VEL
LIN {X 0,Y 448.992,Z 590.601,A -85,B 0,C 180,E1 -8854.571,E2 -8854.571} C_VEL
LIN {X 0,Y 449.316,Z 578.688,A -85,B 0,C 180,E1 -8855.362,E2 -8855.362} C_VEL
LIN {X 0,Y 449.559,Z 566.857,A -85,B 0,C 180,E1 -8855.957,E2 -8855.957} C_VEL
LIN {X 0,Y 449.667,Z 554.456,A -85,B 0,C 180,E1 -8856.401,E2 -8856.401} C_VEL
LIN {X 0,Y 449.681,Z 539.349,A -85,B 0,C 180,E1 -8856.717,E2 -8856.717} C_VEL
LIN {X 0,Y 449.505,Z 529.431,A -85,B 0,C 180,E1 -8856.888,E2 -8856.888} C_VEL
LIN {X 0,Y 446.644,Z 520.722,A -85,B 0,C 180,E1 -8857.147,E2 -8857.147} C_VEL
LIN {X 0,Y 446.448,Z 519.768,A -85,B 0,C 180,E1 -8857.331,E2 -8857.331} C_VEL
LIN {X 0,Y 446.447,Z 519.685,A -85,B 0,C 180,E1 -8860.198,E2 -8860.198} C_VEL
LIN {X 0,Y 446.418,Z 519.692,A -85,B 0,C 180,E1 -8863.601,E2 -8863.601} C_VEL
LIN {X 0,Y 446.445,Z 519.682,A -85,B 0,C 180,E1 -8866.398,E2 -8866.398} C_VEL
LIN {X 0,Y 446.467,Z 519.682,A -85,B 0,C 180,E1 -8869.806,E2 -8869.806} C_VEL
LIN {X 0,Y 446.431,Z 519.684,A -85,B 0,C 180,E1 -8872.125,E2 -8872.125} C_VEL
LIN {X 0,Y 446.429,Z 519.692,A -85,B 0,C 180,E1 -8875.478,E2 -8875.478} C_VEL
LIN {X 0,Y 446.417,Z 519.685,A -85,B 0,C 180,E1 -8878.701,E2 -8878.701} C_VEL
LIN {X 0,Y 446.486,Z 519.68,A -85,B 0,C 180,E1 -8881.822,E2 -8881.822} C_VEL
LIN {X 0,Y 446.459,Z 519.681,A -85,B 0,C 180,E1 -8884.849,E2 -8884.849} C_VEL
LIN {X 0,Y 446.451,Z 519.682,A -85,B 0,C 180,E1 -8888.246,E2 -8888.246} C_VEL
LIN {X 0,Y 446.449,Z 519.681,A -85,B 0,C 180,E1 -8888.553,E2 -8888.553} C_VEL
LIN {X 0,Y 445.795,Z 519.769,A -85,B 0,C 180,E1 -8889.306,E2 -8889.306} C_VEL
LIN {X 0,Y 442.938,Z 520.12,A -85,B 0,C 180,E1 -8890.53,E2 -8890.53} C_VEL
LIN {X 0,Y 440.518,Z 520.427,A -85,B 0,C 180,E1 -8891.517,E2 -8891.517} C_VEL
LIN {X 0,Y 439.487,Z 520.549,A -85,B 0,C 180,E1 -8892.28,E2 -8892.28} C_VEL
LIN {X 0,Y 439.408,Z 520.558,A -85,B 0,C 180,E1 -8892.538,E2 -8892.538} C_VEL
LIN {X 0,Y 439.452,Z 520.555,A -85,B 0,C 180,E1 -8895.175,E2 -8895.175} C_VEL
LIN {X 0,Y 439.488,Z 520.552,A -85,B 0,C 180,E1 -8898.002,E2 -8898.002} C_VEL
LIN {X 0,Y 439.538,Z 520.55,A -85,B 0,C 180,E1 -8901.726,E2 -8901.726} C_VEL
LIN {X 0,Y 439.614,Z 520.533,A -85,B 0,C 180,E1 -8904.496,E2 -8904.496} C_VEL
LIN {X 0,Y 439.639,Z 520.532,A -85,B 0,C 180,E1 -8908.168,E2 -8908.168} C_VEL
LIN {X 0,Y 439.768,Z 520.518,A -85,B 0,C 180,E1 -8910,E2 -8910} C_VEL
LIN {X 0,Y 439.645,Z 520.529,A -85,B 0,C 180,E1 -8912.749,E2 -8912.749} C_VEL
LIN {X 0,Y 439.596,Z 520.536,A -85,B 0,C 180,E1 -8916.425,E2 -8916.425} C_VEL
LIN {X 0,Y 439.501,Z 520.548,A -85,B 0,C 180,E1 -8919.201,E2 -8919.201} C_VEL
LIN {X 0,Y 439.47,Z 520.55,A -85,B 0,C 180,E1 -8922.937,E2 -8922.937} C_VEL
LIN {X 0,Y 439.452,Z 520.555,A -85,B 0,C 180,E1 -8926.348,E2 -8926.348} C_VEL
LIN {X 0,Y 439.406,Z 520.563,A -85,B 0,C 180,E1 -8929.626,E2 -8929.626} C_VEL
LIN {X 0,Y 439.367,Z 520.564,A -85,B 0,C 180,E1 -8932.575,E2 -8932.575} C_VEL
LIN {X 0,Y 439.4,Z 520.563,A -85,B 0,C 180,E1 -8935.585,E2 -8935.585} C_VEL
LIN {X 0,Y 439.419,Z 520.557,A -85,B 0,C 180,E1 -8938.673,E2 -8938.673} C_VEL
LIN {X 0,Y 439.371,Z 520.571,A -85,B 0,C 180,E1 -8942.03,E2 -8942.03} C_VEL
LIN {X 0,Y 439.394,Z 520.561,A -85,B 0,C 180,E1 -8945.339,E2 -8945.339} C_VEL
LIN {X 0,Y 439.395,Z 520.562,A -85,B 0,C 180,E1 -8948.593,E2 -8948.593} C_VEL
LIN {X 0,Y 439.404,Z 520.559,A -85,B 0,C 180,E1 -8951.258,E2 -8951.258} C_VEL
LIN {X 0,Y 439.407,Z 520.56,A -85,B 0,C 180,E1 -8954.727,E2 -8954.727} C_VEL
LIN {X 0,Y 439.393,Z 520.564,A -85,B 0,C 180,E1 -8957.795,E2 -8957.795} C_VEL
LIN {X 0,Y 439.433,Z 520.562,A -85,B 0,C 180,E1 -8960.228,E2 -8960.228} C_VEL
LIN {X 0,Y 439.373,Z 520.565,A -85,B 0,C 180,E1 -8963.712,E2 -8963.712} C_VEL
LIN {X 0,Y 439.371,Z 520.563,A -85,B 0,C 180,E1 -8967.053,E2 -8967.053} C_VEL
LIN {X 0,Y 439.392,Z 520.568,A -85,B 0,C 180,E1 -8970.274,E2 -8970.274} C_VEL
LIN {X 0,Y 439.428,Z 520.557,A -85,B 0,C 180,E1 -8973.588,E2 -8973.588} C_VEL
LIN {X 0,Y 439.381,Z 520.568,A -85,B 0,C 180,E1 -8976.429,E2 -8976.429} C_VEL
LIN {X 0,Y 439.381,Z 520.561,A -85,B 0,C 180,E1 -8979.396,E2 -8979.396} C_VEL
LIN {X 0,Y 439.424,Z 520.564,A -85,B 0,C 180,E1 -8982.309,E2 -8982.309} C_VEL
LIN {X 0,Y 439.439,Z 520.555,A -85,B 0,C 180,E1 -8985.173,E2 -8985.173} C_VEL
LIN {X 0,Y 439.499,Z 520.55,A -85,B 0,C 180,E1 -8988.001,E2 -8988.001} C_VEL
LIN {X 0,Y 439.54,Z 520.542,A -85,B 0,C 180,E1 -8991.726,E2 -8991.726} C_VEL
LIN {X 0,Y 439.618,Z 520.539,A -85,B 0,C 180,E1 -8994.495,E2 -8994.495} C_VEL
LIN {X 0,Y 439.627,Z 520.535,A -85,B 0,C 180,E1 -8998.167,E2 -8998.167} C_VEL
LIN {X 0,Y 439.755,Z 520.517,A -85,B 0,C 180,E1 -9000,E2 -9000} C_VEL
LIN {X 0,Y 439.648,Z 520.533,A -85,B 0,C 180,E1 -9002.748,E2 -9002.748} C_VEL
LIN {X 0,Y 439.609,Z 520.54,A -85,B 0,C 180,E1 -9006.425,E2 -9006.425} C_VEL
LIN {X 0,Y 439.491,Z 520.549,A -85,B 0,C 180,E1 -9009.201,E2 -9009.201} C_VEL
LIN {X 0,Y 439.457,Z 520.556,A -85,B 0,C 180,E1 -9012.938,E2 -9012.938} C_VEL
LIN {X 0,Y 439.439,Z 520.559,A -85,B 0,C 180,E1 -9016.349,E2 -9016.349} C_VEL
LIN {X 0,Y 439.394,Z 520.56,A -85,B 0,C 180,E1 -9019.626,E2 -9019.626} C_VEL
LIN {X 0,Y 439.357,Z 520.571,A -85,B 0,C 180,E1 -9022.576,E2 -9022.576} C_VEL
LIN {X 0,Y 439.397,Z 520.56,A -85,B 0,C 180,E1 -9025.585,E2 -9025.585} C_VEL
LIN {X 0,Y 439.418,Z 520.565,A -85,B 0,C 180,E1 -9028.673,E2 -9028.673} C_VEL
LIN {X 0,Y 439.367,Z 520.563,A -85,B 0,C 180,E1 -9031.861,E2 -9031.861} C_VEL
LIN {X 0,Y 439.394,Z 520.563,A -85,B 0,C 180,E1 -9035.156,E2 -9035.156} C_VEL
LIN {X 0,Y 439.377,Z 520.567,A -85,B 0,C 180,E1 -9038.595,E2 -9038.595} C_VEL
LIN {X 0,Y 439.383,Z 520.564,A -85,B 0,C 180,E1 -9041.257,E2 -9041.257} C_VEL
LIN {X 0,Y 439.401,Z 520.565,A -85,B 0,C 180,E1 -9044.729,E2 -9044.729} C_VEL
LIN {X 0,Y 439.393,Z 520.56,A -85,B 0,C 180,E1 -9047.796,E2 -9047.796} C_VEL
LIN {X 0,Y 439.433,Z 520.556,A -85,B 0,C 180,E1 -9050.229,E2 -9050.229} C_VEL
LIN {X 0,Y 439.373,Z 520.565,A -85,B 0,C 180,E1 -9053.714,E2 -9053.714} C_VEL
LIN {X 0,Y 439.382,Z 520.569,A -85,B 0,C 180,E1 -9057.056,E2 -9057.056} C_VEL
LIN {X 0,Y 439.435,Z 520.619,A -85,B 0,C 180,E1 -9058.039,E2 -9058.039} C_VEL
LIN {X 0,Y 441.157,Z 529.015,A -85,B 0,C 180,E1 -9059.88,E2 -9059.88} C_VEL
LIN {X 0,Y 442.634,Z 537.144,A -85,B 0,C 180,E1 -9061.555,E2 -9061.555} C_VEL
LIN {X 0,Y 441.618,Z 554.872,A -85,B 0,C 180,E1 -9064.937,E2 -9064.937} C_VEL
LIN {X 0,Y 440.657,Z 572.565,A -85,B 0,C 180,E1 -9068.246,E2 -9068.246} C_VEL
LIN {X 0,Y 439.863,Z 589.484,A -85,B 0,C 180,E1 -9071.364,E2 -9071.364} C_VEL
LIN {X 0,Y 439.329,Z 609.056,A -85,B 0,C 180,E1 -9074.933,E2 -9074.933} C_VEL
LIN {X 0,Y 439.266,Z 612.12,A -85,B 0,C 180,E1 -9075.445,E2 -9075.445} C_VEL
LIN {X 0,Y 441.88,Z 643.285,A -85,B 0,C 180,E1 -9076.145,E2 -9076.145} C_VEL
LIN {X 0,Y 441.331,Z 694.146,A -85,B 0,C 180,E1 -9077.118,E2 -9077.118} C_VEL
LIN {X 0,Y 440.874,Z 705.815,A -85,B 0,C 180,E1 -9077.514,E2 -9077.514} C_VEL
LIN {X 0,Y 440.373,Z 718.003,A -85,B 0,C 180,E1 -9078.143,E2 -9078.143} C_VEL
LIN {X 0,Y 439.859,Z 729.24,A -85,B 0,C 180,E1 -9078.946,E2 -9078.946} C_VEL
LIN {X 0,Y 439.433,Z 739.134,A -85,B 0,C 180,E1 -9079.868,E2 -9079.868} C_VEL
LIN {X 0,Y 439.061,Z 747.041,A -85,B 0,C 180,E1 -9080.789,E2 -9080.789} C_VEL
LIN {X 0,Y 438.83,Z 755.019,A -85,B 0,C 180,E1 -9081.945,E2 -9081.945} C_VEL
LIN {X 0,Y 438.766,Z 762.162,A -85,B 0,C 180,E1 -9083.261,E2 -9083.261} C_VEL
LIN {X 0,Y 438.66,Z 767.281,A -85,B 0,C 180,E1 -9084.484,E2 -9084.484} C_VEL
LIN {X 0,Y 438.793,Z 771.656,A -85,B 0,C 180,E1 -9085.867,E2 -9085.867} C_VEL
LIN {X 0,Y 438.753,Z 774.627,A -85,B 0,C 180,E1 -9087.246,E2 -9087.246} C_VEL
LIN {X 0,Y 438.756,Z 775.903,A -85,B 0,C 180,E1 -9088.164,E2 -9088.164} C_VEL
LIN {X 0,Y 438.78,Z 776.641,A -85,B 0,C 180,E1 -9089.082,E2 -9089.082} C_VEL
LIN {X 0,Y 438.97,Z 776.884,A -85,B 0,C 180,E1 -9090,E2 -9090} C_VEL
LIN {X 0,Y 438.796,Z 776.523,A -85,B 0,C 180,E1 -9090.918,E2 -9090.918} C_VEL
LIN {X 0,Y 438.782,Z 775.685,A -85,B 0,C 180,E1 -9091.836,E2 -9091.836} C_VEL
LIN {X 0,Y 438.782,Z 774.278,A -85,B 0,C 180,E1 -9092.754,E2 -9092.754} C_VEL
LIN {X 0,Y 438.813,Z 771.152,A -85,B 0,C 180,E1 -9094.133,E2 -9094.133} C_VEL
LIN {X 0,Y 438.718,Z 766.599,A -85,B 0,C 180,E1 -9095.515,E2 -9095.515} C_VEL
LIN {X 0,Y 438.747,Z 761.414,A -85,B 0,C 180,E1 -9096.718,E2 -9096.718} C_VEL
LIN {X 0,Y 438.801,Z 755.451,A -85,B 0,C 180,E1 -9097.824,E2 -9097.824} C_VEL
LIN {X 0,Y 438.967,Z 747.677,A -85,B 0,C 180,E1 -9098.98,E2 -9098.98} C_VEL
LIN {X 0,Y 439.339,Z 739.012,A -85,B 0,C 180,E1 -9100.018,E2 -9100.018} C_VEL
LIN {X 0,Y 439.739,Z 729.313,A -85,B 0,C 180,E1 -9100.94,E2 -9100.94} C_VEL
LIN {X 0,Y 440.265,Z 718.503,A -85,B 0,C 180,E1 -9101.743,E2 -9101.743} C_VEL
LIN {X 0,Y 440.762,Z 707.276,A -85,B 0,C 180,E1 -9102.372,E2 -9102.372} C_VEL
LIN {X 0,Y 441.266,Z 694.803,A -85,B 0,C 180,E1 -9102.854,E2 -9102.854} C_VEL
LIN {X 0,Y 441.525,Z 682.042,A -85,B 0,C 180,E1 -9103.15,E2 -9103.15} C_VEL
LIN {X 0,Y 441.694,Z 639.547,A -85,B 0,C 180,E1 -9103.929,E2 -9103.929} C_VEL
LIN {X 0,Y 439.212,Z 607.996,A -85,B 0,C 180,E1 -9104.622,E2 -9104.622} C_VEL
LIN {X 0,Y 439.181,Z 606.358,A -85,B 0,C 180,E1 -9104.704,E2 -9104.704} C_VEL
LIN {X 0,Y 439.504,Z 588,A -85,B 0,C 180,E1 -9107.927,E2 -9107.927} C_VEL
LIN {X 0,Y 440.039,Z 570.587,A -85,B 0,C 180,E1 -9111.06,E2 -9111.06} C_VEL
LIN {X 0,Y 440.738,Z 551.977,A -85,B 0,C 180,E1 -9114.493,E2 -9114.493} C_VEL
LIN {X 0,Y 441.605,Z 534.95,A -85,B 0,C 180,E1 -9117.742,E2 -9117.742} C_VEL
LIN {X 0,Y 441.151,Z 529.669,A -85,B 0,C 180,E1 -9118.812,E2 -9118.812} C_VEL
LIN {X 0,Y 439.461,Z 520.678,A -85,B 0,C 180,E1 -9120.78,E2 -9120.78} C_VEL
LIN {X 0,Y 439.384,Z 520.567,A -85,B 0,C 180,E1 -9124.043,E2 -9124.043} C_VEL
LIN {X 0,Y 439.352,Z 520.572,A -85,B 0,C 180,E1 -9126.888,E2 -9126.888} C_VEL
LIN {X 0,Y 439.401,Z 520.561,A -85,B 0,C 180,E1 -9129.849,E2 -9129.849} C_VEL
LIN {X 0,Y 439.381,Z 520.565,A -85,B 0,C 180,E1 -9132.627,E2 -9132.627} C_VEL
LIN {X 0,Y 439.397,Z 520.561,A -85,B 0,C 180,E1 -9136.033,E2 -9136.033} C_VEL
LIN {X 0,Y 439.394,Z 520.567,A -85,B 0,C 180,E1 -9139.021,E2 -9139.021} C_VEL
LIN {X 0,Y 439.386,Z 520.563,A -85,B 0,C 180,E1 -9141.604,E2 -9141.604} C_VEL
LIN {X 0,Y 439.394,Z 520.563,A -85,B 0,C 180,E1 -9144.844,E2 -9144.844} C_VEL
LIN {X 0,Y 439.382,Z 520.561,A -85,B 0,C 180,E1 -9148.141,E2 -9148.141} C_VEL
LIN {X 0,Y 439.417,Z 520.562,A -85,B 0,C 180,E1 -9151.327,E2 -9151.327} C_VEL
LIN {X 0,Y 439.397,Z 520.56,A -85,B 0,C 180,E1 -9154.415,E2 -9154.415} C_VEL
LIN {X 0,Y 439.356,Z 520.569,A -85,B 0,C 180,E1 -9157.424,E2 -9157.424} C_VEL
LIN {X 0,Y 439.432,Z 520.56,A -85,B 0,C 180,E1 -9160.663,E2 -9160.663} C_VEL
LIN {X 0,Y 439.453,Z 520.556,A -85,B 0,C 180,E1 -9164.224,E2 -9164.224} C_VEL
LIN {X 0,Y 439.503,Z 520.549,A -85,B 0,C 180,E1 -9168.002,E2 -9168.002} C_VEL
LIN {X 0,Y 439.538,Z 520.546,A -85,B 0,C 180,E1 -9171.726,E2 -9171.726} C_VEL
LIN {X 0,Y 439.619,Z 520.538,A -85,B 0,C 180,E1 -9174.496,E2 -9174.496} C_VEL
LIN {X 0,Y 439.627,Z 520.536,A -85,B 0,C 180,E1 -9178.168,E2 -9178.168} C_VEL
LIN {X 0,Y 439.755,Z 520.52,A -85,B 0,C 180,E1 -9180,E2 -9180} C_VEL
LIN {X 0,Y 439.649,Z 520.535,A -85,B 0,C 180,E1 -9182.749,E2 -9182.749} C_VEL
LIN {X 0,Y 439.446,Z 520.683,A -85,B 0,C 180,E1 -9184.415,E2 -9184.415} C_VEL
LIN {X 0,Y 439.676,Z 521.633,A -85,B 0,C 180,E1 -9184.584,E2 -9184.584} C_VEL
LIN {X 0,Y 443.081,Z 530.776,A -85,B 0,C 180,E1 -9184.891,E2 -9184.891} C_VEL
LIN {X 0,Y 443.111,Z 554.44,A -85,B 0,C 180,E1 -9185.318,E2 -9185.318} C_VEL
LIN {X 0,Y 443.05,Z 567.793,A -85,B 0,C 180,E1 -9185.747,E2 -9185.747} C_VEL
LIN {X 0,Y 442.908,Z 579.78,A -85,B 0,C 180,E1 -9186.32,E2 -9186.32} C_VEL
LIN {X 0,Y 442.519,Z 591.402,A -85,B 0,C 180,E1 -9187.07,E2 -9187.07} C_VEL
LIN {X 0,Y 442.176,Z 602.453,A -85,B 0,C 180,E1 -9187.995,E2 -9187.995} C_VEL
LIN {X 0,Y 441.708,Z 612.815,A -85,B 0,C 180,E1 -9189.089,E2 -9189.089} C_VEL
LIN {X 0,Y 441.221,Z 622.151,A -85,B 0,C 180,E1 -9190.323,E2 -9190.323} C_VEL
LIN {X 0,Y 440.761,Z 629.37,A -85,B 0,C 180,E1 -9191.497,E2 -9191.497} C_VEL
LIN {X 0,Y 440.377,Z 636.339,A -85,B 0,C 180,E1 -9192.911,E2 -9192.911} C_VEL
LIN {X 0,Y 439.997,Z 641.854,A -85,B 0,C 180,E1 -9194.335,E2 -9194.335} C_VEL
LIN {X 0,Y 439.665,Z 646.122,A -85,B 0,C 180,E1 -9195.768,E2 -9195.768} C_VEL
LIN {X 0,Y 439.518,Z 648.34,A -85,B 0,C 180,E1 -9196.728,E2 -9196.728} C_VEL
LIN {X 0,Y 439.406,Z 650.025,A -85,B 0,C 180,E1 -9197.692,E2 -9197.692} C_VEL
LIN {X 0,Y 439.289,Z 651.82,A -85,B 0,C 180,E1 -9199.284,E2 -9199.284} C_VEL
LIN {X 0,Y 439.175,Z 652.382,A -85,B 0,C 180,E1 -9200.614,E2 -9200.614} C_VEL
LIN {X 0,Y 439.159,Z 652.148,A -85,B 0,C 180,E1 -9201.849,E2 -9201.849} C_VEL
LIN {X 0,Y 439.225,Z 650.56,A -85,B 0,C 180,E1 -9203.58,E2 -9203.58} C_VEL
LIN {X 0,Y 439.387,Z 647.999,A -85,B 0,C 180,E1 -9205.079,E2 -9205.079} C_VEL
LIN {X 0,Y 439.616,Z 644.226,A -85,B 0,C 180,E1 -9206.592,E2 -9206.592} C_VEL
LIN {X 0,Y 439.833,Z 639.269,A -85,B 0,C 180,E1 -9208.061,E2 -9208.061} C_VEL
LIN {X 0,Y 440.161,Z 632.215,A -85,B 0,C 180,E1 -9209.668,E2 -9209.668} C_VEL
LIN {X 0,Y 440.581,Z 625.042,A -85,B 0,C 180,E1 -9210.961,E2 -9210.961} C_VEL
LIN {X 0,Y 440.942,Z 616.988,A -85,B 0,C 180,E1 -9212.143,E2 -9212.143} C_VEL
LIN {X 0,Y 441.446,Z 607.136,A -85,B 0,C 180,E1 -9213.316,E2 -9213.316} C_VEL
LIN {X 0,Y 441.843,Z 597.244,A -85,B 0,C 180,E1 -9214.273,E2 -9214.273} C_VEL
LIN {X 0,Y 442.2,Z 587.448,A -85,B 0,C 180,E1 -9215.04,E2 -9215.04} C_VEL
LIN {X 0,Y 442.524,Z 575.689,A -85,B 0,C 180,E1 -9215.763,E2 -9215.763} C_VEL
LIN {X 0,Y 442.733,Z 562.297,A -85,B 0,C 180,E1 -9216.365,E2 -9216.365} C_VEL
LIN {X 0,Y 442.796,Z 550.281,A -85,B 0,C 180,E1 -9216.726,E2 -9216.726} C_VEL
LIN {X 0,Y 442.75,Z 531.186,A -85,B 0,C 180,E1 -9217.077,E2 -9217.077} C_VEL
LIN {X 0,Y 439.548,Z 521.376,A -85,B 0,C 180,E1 -9217.383,E2 -9217.383} C_VEL
LIN {X 0,Y 439.407,Z 520.621,A -85,B 0,C 180,E1 -9217.574,E2 -9217.574} C_VEL
LIN {X 0,Y 439.409,Z 520.564,A -85,B 0,C 180,E1 -9219.852,E2 -9219.852} C_VEL
LIN {X 0,Y 439.382,Z 520.564,A -85,B 0,C 180,E1 -9222.629,E2 -9222.629} C_VEL
LIN {X 0,Y 439.401,Z 520.56,A -85,B 0,C 180,E1 -9226.035,E2 -9226.035} C_VEL
LIN {X 0,Y 439.399,Z 520.563,A -85,B 0,C 180,E1 -9229.023,E2 -9229.023} C_VEL
LIN {X 0,Y 439.39,Z 520.566,A -85,B 0,C 180,E1 -9231.606,E2 -9231.606} C_VEL
LIN {X 0,Y 439.399,Z 520.561,A -85,B 0,C 180,E1 -9234.845,E2 -9234.845} C_VEL
LIN {X 0,Y 439.373,Z 520.563,A -85,B 0,C 180,E1 -9238.141,E2 -9238.141} C_VEL
LIN {X 0,Y 439.434,Z 520.562,A -85,B 0,C 180,E1 -9241.599,E2 -9241.599} C_VEL
LIN {X 0,Y 439.407,Z 520.558,A -85,B 0,C 180,E1 -9244.416,E2 -9244.416} C_VEL
LIN {X 0,Y 439.368,Z 520.57,A -85,B 0,C 180,E1 -9247.425,E2 -9247.425} C_VEL
LIN {X 0,Y 439.444,Z 520.554,A -85,B 0,C 180,E1 -9250.664,E2 -9250.664} C_VEL
LIN {X 0,Y 439.408,Z 520.558,A -85,B 0,C 180,E1 -9252.538,E2 -9252.538} C_VEL
LIN {X 0,Y 438.748,Z 520.647,A -85,B 0,C 180,E1 -9253.304,E2 -9253.304} C_VEL
LIN {X 0,Y 435.88,Z 520.998,A -85,B 0,C 180,E1 -9254.547,E2 -9254.547} C_VEL
LIN {X 0,Y 433.466,Z 521.306,A -85,B 0,C 180,E1 -9255.55,E2 -9255.55} C_VEL
LIN {X 0,Y 432.455,Z 521.426,A -85,B 0,C 180,E1 -9256.325,E2 -9256.325} C_VEL
LIN {X 0,Y 432.386,Z 521.433,A -85,B 0,C 180,E1 -9256.588,E2 -9256.588} C_VEL
LIN {X 0,Y 432.395,Z 521.432,A -85,B 0,C 180,E1 -9258.753,E2 -9258.753} C_VEL
LIN {X 0,Y 432.487,Z 521.427,A -85,B 0,C 180,E1 -9261.59,E2 -9261.59} C_VEL
LIN {X 0,Y 432.589,Z 521.408,A -85,B 0,C 180,E1 -9264.406,E2 -9264.406} C_VEL
LIN {X 0,Y 432.608,Z 521.408,A -85,B 0,C 180,E1 -9268.138,E2 -9268.138} C_VEL
LIN {X 0,Y 432.737,Z 521.394,A -85,B 0,C 180,E1 -9270,E2 -9270} C_VEL
LIN {X 0,Y 432.597,Z 521.407,A -85,B 0,C 180,E1 -9272.794,E2 -9272.794} C_VEL
LIN {X 0,Y 432.59,Z 521.413,A -85,B 0,C 180,E1 -9275.594,E2 -9275.594} C_VEL
LIN {X 0,Y 432.469,Z 521.424,A -85,B 0,C 180,E1 -9278.41,E2 -9278.41} C_VEL
LIN {X 0,Y 432.464,Z 521.427,A -85,B 0,C 180,E1 -9282.196,E2 -9282.196} C_VEL
LIN {X 0,Y 432.435,Z 521.433,A -85,B 0,C 180,E1 -9286.038,E2 -9286.038} C_VEL
LIN {X 0,Y 432.391,Z 521.435,A -85,B 0,C 180,E1 -9289.485,E2 -9289.485} C_VEL
LIN {X 0,Y 432.321,Z 521.441,A -85,B 0,C 180,E1 -9292.964,E2 -9292.964} C_VEL
LIN {X 0,Y 432.364,Z 521.443,A -85,B 0,C 180,E1 -9296.032,E2 -9296.032} C_VEL
LIN {X 0,Y 432.345,Z 521.438,A -85,B 0,C 180,E1 -9299.187,E2 -9299.187} C_VEL
LIN {X 0,Y 432.324,Z 521.443,A -85,B 0,C 180,E1 -9302.442,E2 -9302.442} C_VEL
LIN {X 0,Y 432.345,Z 521.441,A -85,B 0,C 180,E1 -9305.631,E2 -9305.631} C_VEL
LIN {X 0,Y 432.357,Z 521.437,A -85,B 0,C 180,E1 -9308.716,E2 -9308.716} C_VEL
LIN {X 0,Y 432.373,Z 521.439,A -85,B 0,C 180,E1 -9311.791,E2 -9311.791} C_VEL
LIN {X 0,Y 432.377,Z 521.439,A -85,B 0,C 180,E1 -9314.341,E2 -9314.341} C_VEL
LIN {X 0,Y 432.331,Z 521.447,A -85,B 0,C 180,E1 -9318.202,E2 -9318.202} C_VEL
LIN {X 0,Y 432.349,Z 521.438,A -85,B 0,C 180,E1 -9321.283,E2 -9321.283} C_VEL
LIN {X 0,Y 432.342,Z 521.444,A -85,B 0,C 180,E1 -9324.367,E2 -9324.367} C_VEL
LIN {X 0,Y 432.324,Z 521.442,A -85,B 0,C 180,E1 -9327.557,E2 -9327.557} C_VEL
LIN {X 0,Y 432.39,Z 521.435,A -85,B 0,C 180,E1 -9329.743,E2 -9329.743} C_VEL
LIN {X 0,Y 432.395,Z 521.432,A -85,B 0,C 180,E1 -9333.372,E2 -9333.372} C_VEL
LIN {X 0,Y 432.365,Z 521.44,A -85,B 0,C 180,E1 -9336.023,E2 -9336.023} C_VEL
LIN {X 0,Y 432.343,Z 521.439,A -85,B 0,C 180,E1 -9339.045,E2 -9339.045} C_VEL
LIN {X 0,Y 432.371,Z 521.439,A -85,B 0,C 180,E1 -9342.01,E2 -9342.01} C_VEL
LIN {X 0,Y 432.387,Z 521.434,A -85,B 0,C 180,E1 -9344.926,E2 -9344.926} C_VEL
LIN {X 0,Y 432.473,Z 521.424,A -85,B 0,C 180,E1 -9347.803,E2 -9347.803} C_VEL
LIN {X 0,Y 432.484,Z 521.421,A -85,B 0,C 180,E1 -9351.59,E2 -9351.59} C_VEL
LIN {X 0,Y 432.594,Z 521.415,A -85,B 0,C 180,E1 -9354.406,E2 -9354.406} C_VEL
LIN {X 0,Y 432.597,Z 521.41,A -85,B 0,C 180,E1 -9358.138,E2 -9358.138} C_VEL
LIN {X 0,Y 432.724,Z 521.393,A -85,B 0,C 180,E1 -9360,E2 -9360} C_VEL
LIN {X 0,Y 432.598,Z 521.411,A -85,B 0,C 180,E1 -9362.793,E2 -9362.793} C_VEL
LIN {X 0,Y 432.564,Z 521.419,A -85,B 0,C 180,E1 -9366.53,E2 -9366.53} C_VEL
LIN {X 0,Y 432.434,Z 521.427,A -85,B 0,C 180,E1 -9369.353,E2 -9369.353} C_VEL
LIN {X 0,Y 432.422,Z 521.434,A -85,B 0,C 180,E1 -9372.803,E2 -9372.803} C_VEL
LIN {X 0,Y 432.404,Z 521.437,A -85,B 0,C 180,E1 -9376.479,E2 -9376.479} C_VEL
LIN {X 0,Y 432.331,Z 521.441,A -85,B 0,C 180,E1 -9379.961,E2 -9379.961} C_VEL
LIN {X 0,Y 432.311,Z 521.446,A -85,B 0,C 180,E1 -9382.964,E2 -9382.964} C_VEL
LIN {X 0,Y 432.357,Z 521.437,A -85,B 0,C 180,E1 -9386.033,E2 -9386.033} C_VEL
LIN {X 0,Y 432.345,Z 521.44,A -85,B 0,C 180,E1 -9389.187,E2 -9389.187} C_VEL
LIN {X 0,Y 432.318,Z 521.444,A -85,B 0,C 180,E1 -9392.294,E2 -9392.294} C_VEL
LIN {X 0,Y 432.334,Z 521.446,A -85,B 0,C 180,E1 -9394.677,E2 -9394.677} C_VEL
LIN {X 0,Y 432.339,Z 521.44,A -85,B 0,C 180,E1 -9398.15,E2 -9398.15} C_VEL
LIN {X 0,Y 432.328,Z 521.441,A -85,B 0,C 180,E1 -9401.603,E2 -9401.603} C_VEL
LIN {X 0,Y 432.336,Z 521.441,A -85,B 0,C 180,E1 -9404.347,E2 -9404.347} C_VEL
LIN {X 0,Y 432.32,Z 521.447,A -85,B 0,C 180,E1 -9407.015,E2 -9407.015} C_VEL
LIN {X 0,Y 432.337,Z 521.439,A -85,B 0,C 180,E1 -9409.82,E2 -9409.82} C_VEL
LIN {X 0,Y 432.312,Z 521.449,A -85,B 0,C 180,E1 -9413.023,E2 -9413.023} C_VEL
LIN {X 0,Y 432.356,Z 521.442,A -85,B 0,C 180,E1 -9415.997,E2 -9415.997} C_VEL
LIN {X 0,Y 432.396,Z 521.548,A -85,B 0,C 180,E1 -9417.847,E2 -9417.847} C_VEL
LIN {X 0,Y 434.72,Z 533.089,A -85,B 0,C 180,E1 -9420.38,E2 -9420.38} C_VEL
LIN {X 0,Y 435.671,Z 538.891,A -85,B 0,C 180,E1 -9421.584,E2 -9421.584} C_VEL
LIN {X 0,Y 434.452,Z 558.482,A -85,B 0,C 180,E1 -9425.384,E2 -9425.384} C_VEL
LIN {X 0,Y 433.396,Z 578.043,A -85,B 0,C 180,E1 -9429.099,E2 -9429.099} C_VEL
LIN {X 0,Y 432.596,Z 596.247,A -85,B 0,C 180,E1 -9432.51,E2 -9432.51} C_VEL
LIN {X 0,Y 432.203,Z 610.998,A -85,B 0,C 180,E1 -9435.202,E2 -9435.202} C_VEL
LIN {X 0,Y 434.964,Z 643.39,A -85,B 0,C 180,E1 -9435.947,E2 -9435.947} C_VEL
LIN {X 0,Y 434.353,Z 692.65,A -85,B 0,C 180,E1 -9436.908,E2 -9436.908} C_VEL
LIN {X 0,Y 433.931,Z 704.461,A -85,B 0,C 180,E1 -9437.311,E2 -9437.311} C_VEL
LIN {X 0,Y 433.399,Z 716.719,A -85,B 0,C 180,E1 -9437.949,E2 -9437.949} C_VEL
LIN {X 0,Y 432.927,Z 726.593,A -85,B 0,C 180,E1 -9438.648,E2 -9438.648} C_VEL
LIN {X 0,Y 432.353,Z 736.851,A -85,B 0,C 180,E1 -9439.582,E2 -9439.582} C_VEL
LIN {X 0,Y 432.042,Z 745.901,A -85,B 0,C 180,E1 -9440.638,E2 -9440.638} C_VEL
LIN {X 0,Y 431.775,Z 753.912,A -85,B 0,C 180,E1 -9441.812,E2 -9441.812} C_VEL
LIN {X 0,Y 431.671,Z 760.28,A -85,B 0,C 180,E1 -9442.987,E2 -9442.987} C_VEL
LIN {X 0,Y 431.607,Z 766.227,A -85,B 0,C 180,E1 -9444.393,E2 -9444.393} C_VEL
LIN {X 0,Y 431.734,Z 770.616,A -85,B 0,C 180,E1 -9445.799,E2 -9445.799} C_VEL
LIN {X 0,Y 431.711,Z 773.61,A -85,B 0,C 180,E1 -9447.201,E2 -9447.201} C_VEL
LIN {X 0,Y 431.718,Z 774.89,A -85,B 0,C 180,E1 -9448.134,E2 -9448.134} C_VEL
LIN {X 0,Y 431.747,Z 775.638,A -85,B 0,C 180,E1 -9449.067,E2 -9449.067} C_VEL
LIN {X 0,Y 431.946,Z 775.882,A -85,B 0,C 180,E1 -9450,E2 -9450} C_VEL
LIN {X 0,Y 431.761,Z 775.526,A -85,B 0,C 180,E1 -9450.933,E2 -9450.933} C_VEL
LIN {X 0,Y 431.742,Z 774.685,A -85,B 0,C 180,E1 -9451.866,E2 -9451.866} C_VEL
LIN {X 0,Y 431.737,Z 773.276,A -85,B 0,C 180,E1 -9452.799,E2 -9452.799} C_VEL
LIN {X 0,Y 431.757,Z 770.144,A -85,B 0,C 180,E1 -9454.2,E2 -9454.2} C_VEL
LIN {X 0,Y 431.662,Z 765.584,A -85,B 0,C 180,E1 -9455.606,E2 -9455.606} C_VEL
LIN {X 0,Y 431.65,Z 759.502,A -85,B 0,C 180,E1 -9457.013,E2 -9457.013} C_VEL
LIN {X 0,Y 431.824,Z 751.532,A -85,B 0,C 180,E1 -9458.423,E2 -9458.423} C_VEL
LIN {X 0,Y 432.117,Z 743.051,A -85,B 0,C 180,E1 -9459.596,E2 -9459.596} C_VEL
LIN {X 0,Y 432.476,Z 733.483,A -85,B 0,C 180,E1 -9460.652,E2 -9460.652} C_VEL
LIN {X 0,Y 433.074,Z 722.667,A -85,B 0,C 180,E1 -9461.585,E2 -9461.585} C_VEL
LIN {X 0,Y 433.629,Z 711.05,A -85,B 0,C 180,E1 -9462.341,E2 -9462.341} C_VEL
LIN {X 0,Y 434.16,Z 699.365,A -85,B 0,C 180,E1 -9462.89,E2 -9462.89} C_VEL
LIN {X 0,Y 434.516,Z 686.864,A -85,B 0,C 180,E1 -9463.277,E2 -9463.277} C_VEL
LIN {X 0,Y 434.876,Z 640.416,A -85,B 0,C 180,E1 -9464.152,E2 -9464.152} C_VEL
LIN {X 0,Y 432.224,Z 606.604,A -85,B 0,C 180,E1 -9464.913,E2 -9464.913} C_VEL
LIN {X 0,Y 432.113,Z 604.697,A -85,B 0,C 180,E1 -9465.017,E2 -9465.017} C_VEL
LIN {X 0,Y 432.512,Z 585.433,A -85,B 0,C 180,E1 -9468.473,E2 -9468.473} C_VEL
LIN {X 0,Y 433.094,Z 568.121,A -85,B 0,C 180,E1 -9471.664,E2 -9471.664} C_VEL
LIN {X 0,Y 433.888,Z 549.653,A -85,B 0,C 180,E1 -9475.162,E2 -9475.162} C_VEL
LIN {X 0,Y 434.632,Z 535.349,A -85,B 0,C 180,E1 -9477.964,E2 -9477.964} C_VEL
LIN {X 0,Y 433.825,Z 528.789,A -85,B 0,C 180,E1 -9479.343,E2 -9479.343} C_VEL
LIN {X 0,Y 432.453,Z 521.748,A -85,B 0,C 180,E1 -9480.91,E2 -9480.91} C_VEL
LIN {X 0,Y 432.355,Z 521.443,A -85,B 0,C 180,E1 -9481.342,E2 -9481.342} C_VEL
LIN {X 0,Y 432.337,Z 521.446,A -85,B 0,C 180,E1 -9484.676,E2 -9484.676} C_VEL
LIN {X 0,Y 432.342,Z 521.442,A -85,B 0,C 180,E1 -9488.148,E2 -9488.148} C_VEL
LIN {X 0,Y 432.329,Z 521.442,A -85,B 0,C 180,E1 -9491.602,E2 -9491.602} C_VEL
LIN {X 0,Y 432.337,Z 521.442,A -85,B 0,C 180,E1 -9494.345,E2 -9494.345} C_VEL
LIN {X 0,Y 432.36,Z 521.44,A -85,B 0,C 180,E1 -9497.009,E2 -9497.009} C_VEL
LIN {X 0,Y 432.352,Z 521.439,A -85,B 0,C 180,E1 -9499.816,E2 -9499.816} C_VEL
LIN {X 0,Y 432.311,Z 521.448,A -85,B 0,C 180,E1 -9503.023,E2 -9503.023} C_VEL
LIN {X 0,Y 432.352,Z 521.439,A -85,B 0,C 180,E1 -9505.996,E2 -9505.996} C_VEL
LIN {X 0,Y 432.388,Z 521.434,A -85,B 0,C 180,E1 -9509.744,E2 -9509.744} C_VEL
LIN {X 0,Y 432.392,Z 521.432,A -85,B 0,C 180,E1 -9513.372,E2 -9513.372} C_VEL
LIN {X 0,Y 432.362,Z 521.437,A -85,B 0,C 180,E1 -9516.023,E2 -9516.023} C_VEL
LIN {X 0,Y 432.341,Z 521.442,A -85,B 0,C 180,E1 -9519.046,E2 -9519.046} C_VEL
LIN {X 0,Y 432.369,Z 521.436,A -85,B 0,C 180,E1 -9522.011,E2 -9522.011} C_VEL
LIN {X 0,Y 432.387,Z 521.438,A -85,B 0,C 180,E1 -9524.926,E2 -9524.926} C_VEL
LIN {X 0,Y 432.474,Z 521.425,A -85,B 0,C 180,E1 -9527.804,E2 -9527.804} C_VEL
LIN {X 0,Y 432.483,Z 521.426,A -85,B 0,C 180,E1 -9531.59,E2 -9531.59} C_VEL
LIN {X 0,Y 432.595,Z 521.413,A -85,B 0,C 180,E1 -9534.406,E2 -9534.406} C_VEL
LIN {X 0,Y 432.597,Z 521.412,A -85,B 0,C 180,E1 -9538.138,E2 -9538.138} C_VEL
LIN {X 0,Y 432.725,Z 521.396,A -85,B 0,C 180,E1 -9540,E2 -9540} C_VEL
LIN {X 0,Y 432.599,Z 521.414,A -85,B 0,C 180,E1 -9542.794,E2 -9542.794} C_VEL
LIN {X 0,Y 432.433,Z 521.675,A -85,B 0,C 180,E1 -9544.165,E2 -9544.165} C_VEL
LIN {X 0,Y 432.701,Z 522.777,A -85,B 0,C 180,E1 -9544.308,E2 -9544.308} C_VEL
LIN {X 0,Y 436.258,Z 532.041,A -85,B 0,C 180,E1 -9544.635,E2 -9544.635} C_VEL
LIN {X 0,Y 436.342,Z 556.158,A -85,B 0,C 180,E1 -9545.083,E2 -9545.083} C_VEL
LIN {X 0,Y 436.27,Z 569.351,A -85,B 0,C 180,E1 -9545.518,E2 -9545.518} C_VEL
LIN {X 0,Y 436.092,Z 581.721,A -85,B 0,C 180,E1 -9546.129,E2 -9546.129} C_VEL
LIN {X 0,Y 435.702,Z 593.932,A -85,B 0,C 180,E1 -9546.949,E2 -9546.949} C_VEL
LIN {X 0,Y 435.32,Z 604.715,A -85,B 0,C 180,E1 -9547.888,E2 -9547.888} C_VEL
LIN {X 0,Y 434.787,Z 615.241,A -85,B 0,C 180,E1 -9549.051,E2 -9549.051} C_VEL
LIN {X 0,Y 434.307,Z 623.99,A -85,B 0,C 180,E1 -9550.254,E2 -9550.254} C_VEL
LIN {X 0,Y 433.748,Z 632.286,A -85,B 0,C 180,E1 -9551.686,E2 -9551.686} C_VEL
LIN {X 0,Y 433.342,Z 638.877,A -85,B 0,C 180,E1 -9553.124,E2 -9553.124} C_VEL
LIN {X 0,Y 432.97,Z 644.094,A -85,B 0,C 180,E1 -9554.572,E2 -9554.572} C_VEL
LIN {X 0,Y 432.629,Z 648.067,A -85,B 0,C 180,E1 -9556.032,E2 -9556.032} C_VEL
LIN {X 0,Y 432.485,Z 650.054,A -85,B 0,C 180,E1 -9557.008,E2 -9557.008} C_VEL
LIN {X 0,Y 432.383,Z 651.597,A -85,B 0,C 180,E1 -9557.989,E2 -9557.989} C_VEL
LIN {X 0,Y 432.266,Z 653.009,A -85,B 0,C 180,E1 -9559.443,E2 -9559.443} C_VEL
LIN {X 0,Y 432.166,Z 653.428,A -85,B 0,C 180,E1 -9560.964,E2 -9560.964} C_VEL
LIN {X 0,Y 432.133,Z 653.053,A -85,B 0,C 180,E1 -9562.029,E2 -9562.029} C_VEL
LIN {X 0,Y 432.165,Z 652.299,A -85,B 0,C 180,E1 -9562.973,E2 -9562.973} C_VEL
LIN {X 0,Y 432.283,Z 650.287,A -85,B 0,C 180,E1 -9564.437,E2 -9564.437} C_VEL
LIN {X 0,Y 432.495,Z 646.908,A -85,B 0,C 180,E1 -9566.024,E2 -9566.024} C_VEL
LIN {X 0,Y 432.73,Z 642.282,A -85,B 0,C 180,E1 -9567.573,E2 -9567.573} C_VEL
LIN {X 0,Y 433.025,Z 636.149,A -85,B 0,C 180,E1 -9569.137,E2 -9569.137} C_VEL
LIN {X 0,Y 433.43,Z 629.486,A -85,B 0,C 180,E1 -9570.48,E2 -9570.48} C_VEL
LIN {X 0,Y 433.862,Z 621.568,A -85,B 0,C 180,E1 -9571.767,E2 -9571.767} C_VEL
LIN {X 0,Y 434.328,Z 612.795,A -85,B 0,C 180,E1 -9572.931,E2 -9572.931} C_VEL
LIN {X 0,Y 434.716,Z 602.548,A -85,B 0,C 180,E1 -9574.041,E2 -9574.041} C_VEL
LIN {X 0,Y 435.22,Z 591.318,A -85,B 0,C 180,E1 -9575,E2 -9575} C_VEL
LIN {X 0,Y 435.536,Z 580.059,A -85,B 0,C 180,E1 -9575.756,E2 -9575.756} C_VEL
LIN {X 0,Y 435.8,Z 567.659,A -85,B 0,C 180,E1 -9576.386,E2 -9576.386} C_VEL
LIN {X 0,Y 435.854,Z 554.404,A -85,B 0,C 180,E1 -9576.845,E2 -9576.845} C_VEL
LIN {X 0,Y 435.716,Z 532.168,A -85,B 0,C 180,E1 -9577.287,E2 -9577.287} C_VEL
LIN {X 0,Y 432.546,Z 522.396,A -85,B 0,C 180,E1 -9577.592,E2 -9577.592} C_VEL
LIN {X 0,Y 432.39,Z 521.533,A -85,B 0,C 180,E1 -9577.765,E2 -9577.765} C_VEL
LIN {X 0,Y 432.325,Z 521.445,A -85,B 0,C 180,E1 -9580.561,E2 -9580.561} C_VEL
LIN {X 0,Y 432.32,Z 521.446,A -85,B 0,C 180,E1 -9583.061,E2 -9583.061} C_VEL
LIN {X 0,Y 432.376,Z 521.438,A -85,B 0,C 180,E1 -9585.66,E2 -9585.66} C_VEL
LIN {X 0,Y 432.371,Z 521.435,A -85,B 0,C 180,E1 -9588.393,E2 -9588.393} C_VEL
LIN {X 0,Y 432.351,Z 521.44,A -85,B 0,C 180,E1 -9591.853,E2 -9591.853} C_VEL
LIN {X 0,Y 432.34,Z 521.445,A -85,B 0,C 180,E1 -9595.324,E2 -9595.324} C_VEL
LIN {X 0,Y 432.322,Z 521.441,A -85,B 0,C 180,E1 -9598.655,E2 -9598.655} C_VEL
LIN {X 0,Y 432.384,Z 521.436,A -85,B 0,C 180,E1 -9601.878,E2 -9601.878} C_VEL
LIN {X 0,Y 432.354,Z 521.439,A -85,B 0,C 180,E1 -9605,E2 -9605} C_VEL
LIN {X 0,Y 432.36,Z 521.438,A -85,B 0,C 180,E1 -9608.047,E2 -9608.047} C_VEL
LIN {X 0,Y 432.388,Z 521.434,A -85,B 0,C 180,E1 -9611.03,E2 -9611.03} C_VEL
LIN {X 0,Y 432.434,Z 521.43,A -85,B 0,C 180,E1 -9613.962,E2 -9613.962} C_VEL
LIN {X 0,Y 432.386,Z 521.433,A -85,B 0,C 180,E1 -9616.588,E2 -9616.588} C_VEL
LIN {X 0,Y 431.759,Z 521.518,A -85,B 0,C 180,E1 -9617.365,E2 -9617.365} C_VEL
LIN {X 0,Y 428.929,Z 521.864,A -85,B 0,C 180,E1 -9618.628,E2 -9618.628} C_VEL
LIN {X 0,Y 426.516,Z 522.172,A -85,B 0,C 180,E1 -9619.647,E2 -9619.647} C_VEL
LIN {X 0,Y 425.483,Z 522.294,A -85,B 0,C 180,E1 -9620.435,E2 -9620.435} C_VEL
LIN {X 0,Y 425.402,Z 522.303,A -85,B 0,C 180,E1 -9620.702,E2 -9620.702} C_VEL
LIN {X 0,Y 425.502,Z 522.294,A -85,B 0,C 180,E1 -9623.361,E2 -9623.361} C_VEL
LIN {X 0,Y 425.369,Z 522.31,A -85,B 0,C 180,E1 -9625.262,E2 -9625.262} C_VEL
LIN {X 0,Y 425.578,Z 522.284,A -85,B 0,C 180,E1 -9628.107,E2 -9628.107} C_VEL
LIN {X 0,Y 425.707,Z 522.269,A -85,B 0,C 180,E1 -9630,E2 -9630} C_VEL
LIN {X 0,Y 425.55,Z 522.284,A -85,B 0,C 180,E1 -9632.84,E2 -9632.84} C_VEL
LIN {X 0,Y 425.545,Z 522.292,A -85,B 0,C 180,E1 -9635.687,E2 -9635.687} C_VEL
LIN {X 0,Y 425.413,Z 522.302,A -85,B 0,C 180,E1 -9638.551,E2 -9638.551} C_VEL
LIN {X 0,Y 425.417,Z 522.303,A -85,B 0,C 180,E1 -9642.401,E2 -9642.401} C_VEL
LIN {X 0,Y 425.393,Z 522.307,A -85,B 0,C 180,E1 -9646.311,E2 -9646.311} C_VEL
LIN {X 0,Y 425.332,Z 522.316,A -85,B 0,C 180,E1 -9649.635,E2 -9649.635} C_VEL
LIN {X 0,Y 425.291,Z 522.32,A -85,B 0,C 180,E1 -9652.338,E2 -9652.338} C_VEL
LIN {X 0,Y 425.293,Z 522.318,A -85,B 0,C 180,E1 -9655.445,E2 -9655.445} C_VEL
LIN {X 0,Y 425.35,Z 522.312,A -85,B 0,C 180,E1 -9657.557,E2 -9657.557} C_VEL
LIN {X 0,Y 425.289,Z 522.317,A -85,B 0,C 180,E1 -9660.815,E2 -9660.815} C_VEL
LIN {X 0,Y 425.312,Z 522.319,A -85,B 0,C 180,E1 -9664.287,E2 -9664.287} C_VEL
LIN {X 0,Y 425.287,Z 522.321,A -85,B 0,C 180,E1 -9667.692,E2 -9667.692} C_VEL
LIN {X 0,Y 425.301,Z 522.318,A -85,B 0,C 180,E1 -9670.523,E2 -9670.523} C_VEL
LIN {X 0,Y 425.315,Z 522.314,A -85,B 0,C 180,E1 -9673.358,E2 -9673.358} C_VEL
LIN {X 0,Y 425.256,Z 522.323,A -85,B 0,C 180,E1 -9676.648,E2 -9676.648} C_VEL
LIN {X 0,Y 425.292,Z 522.321,A -85,B 0,C 180,E1 -9679.873,E2 -9679.873} C_VEL
LIN {X 0,Y 425.281,Z 522.322,A -85,B 0,C 180,E1 -9682.486,E2 -9682.486} C_VEL
LIN {X 0,Y 425.304,Z 522.318,A -85,B 0,C 180,E1 -9685.816,E2 -9685.816} C_VEL
LIN {X 0,Y 425.299,Z 522.316,A -85,B 0,C 180,E1 -9689.235,E2 -9689.235} C_VEL
LIN {X 0,Y 425.345,Z 522.315,A -85,B 0,C 180,E1 -9692.442,E2 -9692.442} C_VEL
LIN {X 0,Y 425.345,Z 522.311,A -85,B 0,C 180,E1 -9695.601,E2 -9695.601} C_VEL
LIN {X 0,Y 425.286,Z 522.321,A -85,B 0,C 180,E1 -9698.681,E2 -9698.681} C_VEL
LIN {X 0,Y 425.326,Z 522.313,A -85,B 0,C 180,E1 -9701.702,E2 -9701.702} C_VEL
LIN {X 0,Y 425.341,Z 522.314,A -85,B 0,C 180,E1 -9704.67,E2 -9704.67} C_VEL
LIN {X 0,Y 425.422,Z 522.301,A -85,B 0,C 180,E1 -9707.598,E2 -9707.598} C_VEL
LIN {X 0,Y 425.435,Z 522.299,A -85,B 0,C 180,E1 -9711.449,E2 -9711.449} C_VEL
LIN {X 0,Y 425.551,Z 522.291,A -85,B 0,C 180,E1 -9714.313,E2 -9714.313} C_VEL
LIN {X 0,Y 425.567,Z 522.286,A -85,B 0,C 180,E1 -9718.107,E2 -9718.107} C_VEL
LIN {X 0,Y 425.694,Z 522.269,A -85,B 0,C 180,E1 -9720,E2 -9720} C_VEL
LIN {X 0,Y 425.549,Z 522.288,A -85,B 0,C 180,E1 -9722.84,E2 -9722.84} C_VEL
LIN {X 0,Y 425.521,Z 522.295,A -85,B 0,C 180,E1 -9726.639,E2 -9726.639} C_VEL
LIN {X 0,Y 425.393,Z 522.304,A -85,B 0,C 180,E1 -9729.509,E2 -9729.509} C_VEL
LIN {X 0,Y 425.385,Z 522.309,A -85,B 0,C 180,E1 -9732.904,E2 -9732.904} C_VEL
LIN {X 0,Y 425.353,Z 522.317,A -85,B 0,C 180,E1 -9736.605,E2 -9736.605} C_VEL
LIN {X 0,Y 425.32,Z 522.313,A -85,B 0,C 180,E1 -9739.636,E2 -9739.636} C_VEL
LIN {X 0,Y 425.28,Z 522.322,A -85,B 0,C 180,E1 -9742.339,E2 -9742.339} C_VEL
LIN {X 0,Y 425.287,Z 522.318,A -85,B 0,C 180,E1 -9745.446,E2 -9745.446} C_VEL
LIN {X 0,Y 425.33,Z 522.319,A -85,B 0,C 180,E1 -9748.632,E2 -9748.632} C_VEL
LIN {X 0,Y 425.259,Z 522.321,A -85,B 0,C 180,E1 -9751.927,E2 -9751.927} C_VEL
LIN {X 0,Y 425.294,Z 522.318,A -85,B 0,C 180,E1 -9755.336,E2 -9755.336} C_VEL
LIN {X 0,Y 425.303,Z 522.322,A -85,B 0,C 180,E1 -9758.898,E2 -9758.898} C_VEL
LIN {X 0,Y 425.286,Z 522.318,A -85,B 0,C 180,E1 -9761.959,E2 -9761.959} C_VEL
LIN {X 0,Y 425.286,Z 522.32,A -85,B 0,C 180,E1 -9765.283,E2 -9765.283} C_VEL
LIN {X 0,Y 425.272,Z 522.324,A -85,B 0,C 180,E1 -9768.622,E2 -9768.622} C_VEL
LIN {X 0,Y 425.312,Z 522.319,A -85,B 0,C 180,E1 -9771.104,E2 -9771.104} C_VEL
LIN {X 0,Y 425.297,Z 522.323,A -85,B 0,C 180,E1 -9774.665,E2 -9774.665} C_VEL
LIN {X 0,Y 425.326,Z 522.426,A -85,B 0,C 180,E1 -9777.632,E2 -9777.632} C_VEL
LIN {X 0,Y 427.93,Z 535.353,A -85,B 0,C 180,E1 -9780.508,E2 -9780.508} C_VEL
LIN {X 0,Y 428.671,Z 540.59,A -85,B 0,C 180,E1 -9781.612,E2 -9781.612} C_VEL
LIN {X 0,Y 427.392,Z 560.127,A -85,B 0,C 180,E1 -9785.468,E2 -9785.468} C_VEL
LIN {X 0,Y 426.234,Z 579.593,A -85,B 0,C 180,E1 -9789.237,E2 -9789.237} C_VEL
LIN {X 0,Y 425.533,Z 596.451,A -85,B 0,C 180,E1 -9792.458,E2 -9792.458} C_VEL
LIN {X 0,Y 425.148,Z 609.673,A -85,B 0,C 180,E1 -9794.933,E2 -9794.933} C_VEL
LIN {X 0,Y 425.791,Z 617.912,A -85,B 0,C 180,E1 -9795.159,E2 -9795.159} C_VEL
LIN {X 0,Y 428.038,Z 644.581,A -85,B 0,C 180,E1 -9795.764,E2 -9795.764} C_VEL
LIN {X 0,Y 427.41,Z 692.205,A -85,B 0,C 180,E1 -9796.721,E2 -9796.721} C_VEL
LIN {X 0,Y 427.004,Z 703.093,A -85,B 0,C 180,E1 -9797.102,E2 -9797.102} C_VEL
LIN {X 0,Y 426.522,Z 713.482,A -85,B 0,C 180,E1 -9797.631,E2 -9797.631} C_VEL
LIN {X 0,Y 426.075,Z 723.902,A -85,B 0,C 180,E1 -9798.343,E2 -9798.343} C_VEL
LIN {X 0,Y 425.521,Z 733.32,A -85,B 0,C 180,E1 -9799.172,E2 -9799.172} C_VEL
LIN {X 0,Y 425.04,Z 742.932,A -85,B 0,C 180,E1 -9800.242,E2 -9800.242} C_VEL
LIN {X 0,Y 424.751,Z 751.327,A -85,B 0,C 180,E1 -9801.436,E2 -9801.436} C_VEL
LIN {X 0,Y 424.579,Z 758.156,A -85,B 0,C 180,E1 -9802.654,E2 -9802.654} C_VEL
LIN {X 0,Y 424.612,Z 763.852,A -85,B 0,C 180,E1 -9803.948,E2 -9803.948} C_VEL
LIN {X 0,Y 424.606,Z 768.275,A -85,B 0,C 180,E1 -9805.253,E2 -9805.253} C_VEL
LIN {X 0,Y 424.732,Z 770.73,A -85,B 0,C 180,E1 -9806.205,E2 -9806.205} C_VEL
LIN {X 0,Y 424.669,Z 772.593,A -85,B 0,C 180,E1 -9807.154,E2 -9807.154} C_VEL
LIN {X 0,Y 424.68,Z 773.876,A -85,B 0,C 180,E1 -9808.103,E2 -9808.103} C_VEL
LIN {X 0,Y 424.714,Z 774.635,A -85,B 0,C 180,E1 -9809.052,E2 -9809.052} C_VEL
LIN {X 0,Y 424.923,Z 774.88,A -85,B 0,C 180,E1 -9810,E2 -9810} C_VEL
LIN {X 0,Y 424.727,Z 774.527,A -85,B 0,C 180,E1 -9810.948,E2 -9810.948} C_VEL
LIN {X 0,Y 424.701,Z 773.683,A -85,B 0,C 180,E1 -9811.897,E2 -9811.897} C_VEL
LIN {X 0,Y 424.692,Z 772.271,A -85,B 0,C 180,E1 -9812.846,E2 -9812.846} C_VEL
LIN {X 0,Y 424.687,Z 769.133,A -85,B 0,C 180,E1 -9814.271,E2 -9814.271} C_VEL
LIN {X 0,Y 424.608,Z 764.581,A -85,B 0,C 180,E1 -9815.699,E2 -9815.699} C_VEL
LIN {X 0,Y 424.557,Z 758.511,A -85,B 0,C 180,E1 -9817.131,E2 -9817.131} C_VEL
LIN {X 0,Y 424.751,Z 750.565,A -85,B 0,C 180,E1 -9818.564,E2 -9818.564} C_VEL
LIN {X 0,Y 425.044,Z 742.115,A -85,B 0,C 180,E1 -9819.757,E2 -9819.757} C_VEL
LIN {X 0,Y 425.494,Z 732.599,A -85,B 0,C 180,E1 -9820.829,E2 -9820.829} C_VEL
LIN {X 0,Y 426.1,Z 721.83,A -85,B 0,C 180,E1 -9821.777,E2 -9821.777} C_VEL
LIN {X 0,Y 426.644,Z 711.346,A -85,B 0,C 180,E1 -9822.486,E2 -9822.486} C_VEL
LIN {X 0,Y 427.214,Z 699.659,A -85,B 0,C 180,E1 -9823.073,E2 -9823.073} C_VEL
LIN {X 0,Y 427.619,Z 686.974,A -85,B 0,C 180,E1 -9823.494,E2 -9823.494} C_VEL
LIN {X 0,Y 428.012,Z 640.613,A -85,B 0,C 180,E1 -9824.4,E2 -9824.4} C_VEL
LIN {X 0,Y 425.463,Z 607.353,A -85,B 0,C 180,E1 -9825.173,E2 -9825.173} C_VEL
LIN {X 0,Y 425.066,Z 603.177,A -85,B 0,C 180,E1 -9825.322,E2 -9825.322} C_VEL
LIN {X 0,Y 425.431,Z 585.571,A -85,B 0,C 180,E1 -9828.542,E2 -9828.542} C_VEL
LIN {X 0,Y 426.05,Z 568.342,A -85,B 0,C 180,E1 -9831.786,E2 -9831.786} C_VEL
LIN {X 0,Y 426.896,Z 549.976,A -85,B 0,C 180,E1 -9835.342,E2 -9835.342} C_VEL
LIN {X 0,Y 427.65,Z 535.759,A -85,B 0,C 180,E1 -9838.194,E2 -9838.194} C_VEL
LIN {X 0,Y 426.185,Z 526.625,A -85,B 0,C 180,E1 -9840.195,E2 -9840.195} C_VEL
LIN {X 0,Y 425.344,Z 522.385,A -85,B 0,C 180,E1 -9841.224,E2 -9841.224} C_VEL
LIN {X 0,Y 425.308,Z 522.321,A -85,B 0,C 180,E1 -9844.287,E2 -9844.287} C_VEL
LIN {X 0,Y 425.281,Z 522.322,A -85,B 0,C 180,E1 -9847.693,E2 -9847.693} C_VEL
LIN {X 0,Y 425.277,Z 522.322,A -85,B 0,C 180,E1 -9850.52,E2 -9850.52} C_VEL
LIN {X 0,Y 425.259,Z 522.326,A -85,B 0,C 180,E1 -9853.351,E2 -9853.351} C_VEL
LIN {X 0,Y 425.326,Z 522.318,A -85,B 0,C 180,E1 -9856.638,E2 -9856.638} C_VEL
LIN {X 0,Y 425.305,Z 522.317,A -85,B 0,C 180,E1 -9859.875,E2 -9859.875} C_VEL
LIN {X 0,Y 425.28,Z 522.322,A -85,B 0,C 180,E1 -9862.486,E2 -9862.486} C_VEL
LIN {X 0,Y 425.3,Z 522.318,A -85,B 0,C 180,E1 -9865.817,E2 -9865.817} C_VEL
LIN {X 0,Y 425.298,Z 522.32,A -85,B 0,C 180,E1 -9869.235,E2 -9869.235} C_VEL
LIN {X 0,Y 425.342,Z 522.315,A -85,B 0,C 180,E1 -9872.442,E2 -9872.442} C_VEL
LIN {X 0,Y 425.342,Z 522.313,A -85,B 0,C 180,E1 -9875.602,E2 -9875.602} C_VEL
LIN {X 0,Y 425.284,Z 522.325,A -85,B 0,C 180,E1 -9878.681,E2 -9878.681} C_VEL
LIN {X 0,Y 425.324,Z 522.314,A -85,B 0,C 180,E1 -9881.703,E2 -9881.703} C_VEL
LIN {X 0,Y 425.339,Z 522.315,A -85,B 0,C 180,E1 -9884.671,E2 -9884.671} C_VEL
LIN {X 0,Y 425.423,Z 522.304,A -85,B 0,C 180,E1 -9887.599,E2 -9887.599} C_VEL
LIN {X 0,Y 425.433,Z 522.305,A -85,B 0,C 180,E1 -9891.45,E2 -9891.45} C_VEL
LIN {X 0,Y 425.57,Z 522.288,A -85,B 0,C 180,E1 -9894.314,E2 -9894.314} C_VEL
LIN {X 0,Y 425.567,Z 522.287,A -85,B 0,C 180,E1 -9898.108,E2 -9898.108} C_VEL
LIN {X 0,Y 425.695,Z 522.272,A -85,B 0,C 180,E1 -9900,E2 -9900} C_VEL
LIN {X 0,Y 425.551,Z 522.292,A -85,B 0,C 180,E1 -9902.84,E2 -9902.84} C_VEL
LIN {X 0,Y 425.409,Z 522.597,A -85,B 0,C 180,E1 -9903.878,E2 -9903.878} C_VEL
LIN {X 0,Y 425.731,Z 523.894,A -85,B 0,C 180,E1 -9904.023,E2 -9904.023} C_VEL
LIN {X 0,Y 429.431,Z 533.446,A -85,B 0,C 180,E1 -9904.369,E2 -9904.369} C_VEL
LIN {X 0,Y 429.562,Z 557.911,A -85,B 0,C 180,E1 -9904.84,E2 -9904.84} C_VEL
LIN {X 0,Y 429.526,Z 570.868,A -85,B 0,C 180,E1 -9905.281,E2 -9905.281} C_VEL
LIN {X 0,Y 429.328,Z 582.666,A -85,B 0,C 180,E1 -9905.873,E2 -9905.873} C_VEL
LIN {X 0,Y 428.923,Z 594.925,A -85,B 0,C 180,E1 -9906.705,E2 -9906.705} C_VEL
LIN {X 0,Y 428.521,Z 605.751,A -85,B 0,C 180,E1 -9907.658,E2 -9907.658} C_VEL
LIN {X 0,Y 428.021,Z 615.268,A -85,B 0,C 180,E1 -9908.711,E2 -9908.711} C_VEL
LIN {X 0,Y 427.524,Z 623.934,A -85,B 0,C 180,E1 -9909.892,E2 -9909.892} C_VEL
LIN {X 0,Y 426.995,Z 631.479,A -85,B 0,C 180,E1 -9911.151,E2 -9911.151} C_VEL
LIN {X 0,Y 426.543,Z 638.46,A -85,B 0,C 180,E1 -9912.611,E2 -9912.611} C_VEL
LIN {X 0,Y 426.179,Z 643,A -85,B 0,C 180,E1 -9913.786,E2 -9913.786} C_VEL
LIN {X 0,Y 425.787,Z 647.612,A -85,B 0,C 180,E1 -9915.314,E2 -9915.314} C_VEL
LIN {X 0,Y 425.525,Z 650.683,A -85,B 0,C 180,E1 -9916.683,E2 -9916.683} C_VEL
LIN {X 0,Y 425.333,Z 653.081,A -85,B 0,C 180,E1 -9918.298,E2 -9918.298} C_VEL
LIN {X 0,Y 425.223,Z 654.152,A -85,B 0,C 180,E1 -9919.599,E2 -9919.599} C_VEL
LIN {X 0,Y 425.119,Z 654.359,A -85,B 0,C 180,E1 -9921.328,E2 -9921.328} C_VEL
LIN {X 0,Y 425.133,Z 653.869,A -85,B 0,C 180,E1 -9922.348,E2 -9922.348} C_VEL
LIN {X 0,Y 425.174,Z 652.865,A -85,B 0,C 180,E1 -9923.373,E2 -9923.373} C_VEL
LIN {X 0,Y 425.296,Z 650.96,A -85,B 0,C 180,E1 -9924.653,E2 -9924.653} C_VEL
LIN {X 0,Y 425.459,Z 648.184,A -85,B 0,C 180,E1 -9925.96,E2 -9925.96} C_VEL
LIN {X 0,Y 425.719,Z 643.65,A -85,B 0,C 180,E1 -9927.532,E2 -9927.532} C_VEL
LIN {X 0,Y 426.002,Z 637.979,A -85,B 0,C 180,E1 -9929.032,E2 -9929.032} C_VEL
LIN {X 0,Y 426.404,Z 631.199,A -85,B 0,C 180,E1 -9930.453,E2 -9930.453} C_VEL
LIN {X 0,Y 426.865,Z 623.26,A -85,B 0,C 180,E1 -9931.794,E2 -9931.794} C_VEL
LIN {X 0,Y 427.351,Z 614.445,A -85,B 0,C 180,E1 -9932.997,E2 -9932.997} C_VEL
LIN {X 0,Y 427.764,Z 604.584,A -85,B 0,C 180,E1 -9934.097,E2 -9934.097} C_VEL
LIN {X 0,Y 428.244,Z 593.873,A -85,B 0,C 180,E1 -9935.058,E2 -9935.058} C_VEL
LIN {X 0,Y 428.619,Z 581.994,A -85,B 0,C 180,E1 -9935.887,E2 -9935.887} C_VEL
LIN {X 0,Y 428.883,Z 569.639,A -85,B 0,C 180,E1 -9936.539,E2 -9936.539} C_VEL
LIN {X 0,Y 428.996,Z 557.373,A -85,B 0,C 180,E1 -9936.994,E2 -9936.994} C_VEL
LIN {X 0,Y 429.05,Z 540.896,A -85,B 0,C 180,E1 -9937.35,E2 -9937.35} C_VEL
LIN {X 0,Y 428.974,Z 533.954,A -85,B 0,C 180,E1 -9937.476,E2 -9937.476} C_VEL
LIN {X 0,Y 425.529,Z 523.426,A -85,B 0,C 180,E1 -9937.801,E2 -9937.801} C_VEL
LIN {X 0,Y 425.341,Z 522.481,A -85,B 0,C 180,E1 -9937.954,E2 -9937.954} C_VEL
LIN {X 0,Y 425.273,Z 522.326,A -85,B 0,C 180,E1 -9941.379,E2 -9941.379} C_VEL
LIN {X 0,Y 425.297,Z 522.317,A -85,B 0,C 180,E1 -9944.72,E2 -9944.72} C_VEL
LIN {X 0,Y 425.342,Z 522.311,A -85,B 0,C 180,E1 -9948.035,E2 -9948.035} C_VEL
LIN {X 0,Y 425.322,Z 522.317,A -85,B 0,C 180,E1 -9951.105,E2 -9951.105} C_VEL
LIN {X 0,Y 425.299,Z 522.316,A -85,B 0,C 180,E1 -9954.665,E2 -9954.665} C_VEL
LIN {X 0,Y 425.265,Z 522.321,A -85,B 0,C 180,E1 -9958.074,E2 -9958.074} C_VEL
LIN {X 0,Y 425.333,Z 522.318,A -85,B 0,C 180,E1 -9961.369,E2 -9961.369} C_VEL
LIN {X 0,Y 425.297,Z 522.316,A -85,B 0,C 180,E1 -9964.556,E2 -9964.556} C_VEL
LIN {X 0,Y 425.29,Z 522.323,A -85,B 0,C 180,E1 -9967.662,E2 -9967.662} C_VEL
LIN {X 0,Y 425.364,Z 522.308,A -85,B 0,C 180,E1 -9970.705,E2 -9970.705} C_VEL
LIN {X 0,Y 425.391,Z 522.311,A -85,B 0,C 180,E1 -9973.689,E2 -9973.689} C_VEL
LIN {X 0,Y 425.416,Z 522.309,A -85,B 0,C 180,E1 -9977.599,E2 -9977.599} C_VEL
LIN {X 0,Y 425.402,Z 522.303,A -85,B 0,C 180,E1 -9980.702,E2 -9980.702} C_VEL
LIN {X 0,Y 424.763,Z 522.388,A -85,B 0,C 180,E1 -9981.493,E2 -9981.493} C_VEL
LIN {X 0,Y 421.976,Z 522.73,A -85,B 0,C 180,E1 -9982.779,E2 -9982.779} C_VEL
LIN {X 0,Y 419.574,Z 523.035,A -85,B 0,C 180,E1 -9983.817,E2 -9983.817} C_VEL
LIN {X 0,Y 418.491,Z 523.165,A -85,B 0,C 180,E1 -9984.619,E2 -9984.619} C_VEL
LIN {X 0,Y 418.376,Z 523.179,A -85,B 0,C 180,E1 -9984.89,E2 -9984.89} C_VEL
LIN {X 0,Y 418.547,Z 523.16,A -85,B 0,C 180,E1 -9988.076,E2 -9988.076} C_VEL
LIN {X 0,Y 418.676,Z 523.145,A -85,B 0,C 180,E1 -9990,E2 -9990} C_VEL
LIN {X 0,Y 418.506,Z 523.162,A -85,B 0,C 180,E1 -9992.888,E2 -9992.888} C_VEL
LIN {X 0,Y 418.503,Z 523.17,A -85,B 0,C 180,E1 -9995.783,E2 -9995.783} C_VEL
LIN {X 0,Y 418.382,Z 523.177,A -85,B 0,C 180,E1 -9998.695,E2 -9998.695} C_VEL
LIN {X 0,Y 418.32,Z 523.19,A -85,B 0,C 180,E1 -10001.631,E2 -10001.631} C_VEL
LIN {X 0,Y 418.307,Z 523.187,A -85,B 0,C 180,E1 -10004.597,E2 -10004.597} C_VEL
LIN {X 0,Y 418.292,Z 523.193,A -85,B 0,C 180,E1 -10007.603,E2 -10007.603} C_VEL
LIN {X 0,Y 418.253,Z 523.194,A -85,B 0,C 180,E1 -10010.662,E2 -10010.662} C_VEL
LIN {X 0,Y 418.277,Z 523.196,A -85,B 0,C 180,E1 -10013.781,E2 -10013.781} C_VEL
LIN {X 0,Y 418.312,Z 523.186,A -85,B 0,C 180,E1 -10017.07,E2 -10017.07} C_VEL
LIN {X 0,Y 418.246,Z 523.199,A -85,B 0,C 180,E1 -10020.271,E2 -10020.271} C_VEL
LIN {X 0,Y 418.249,Z 523.198,A -85,B 0,C 180,E1 -10023.676,E2 -10023.676} C_VEL
